	LOCAL CONST Robtarget Tr_meulage_bavure_P179 :=[[-62.25637890625,114.8428984375,23],[0.0433975001230337,-0.0506645555826487,0.757781496955649,-0.649089333345064],[0,0,0,0],[8.999999E+09,8.999999E+09,8.999999E+09,8.999999E+09,8.999999E+09,8.999999E+09]];
	LOCAL CONST Robtarget Tr_meulage_bavure_P180 :=[[-59.10421875,115.2802421875,23],[0.0426624400154122,-0.0495768426742355,0.75636290662596,-0.650874186277744],[0,0,0,0],[8.999999E+09,8.999999E+09,8.999999E+09,8.999999E+09,8.999999E+09,8.999999E+09]];
	LOCAL CONST Robtarget Tr_meulage_bavure_P181 :=[[-53.5016484375,115.9119296875,23],[0.0425676623921922,-0.0492400718100533,0.754898413474392,-0.652603857466726],[0,0,0,0],[8.999999E+09,8.999999E+09,8.999999E+09,8.999999E+09,8.999999E+09,8.999999E+09]];
	LOCAL CONST Robtarget Tr_meulage_bavure_P182 :=[[-50.74237109375,116.2019375,23],[0.0427141238515756,-0.0491877810931781,0.753441246798892,-0.654280026775121],[0,0,0,0],[8.999999E+09,8.999999E+09,8.999999E+09,8.999999E+09,8.999999E+09,8.999999E+09]];
	LOCAL CONST Robtarget Tr_meulage_bavure_P183 :=[[-48.3789375,116.5492578125,23],[0.0426883692327484,-0.0489442555493909,0.752036641826874,-0.65591390618794],[0,0,0,0],[8.999999E+09,8.999999E+09,8.999999E+09,8.999999E+09,8.999999E+09,8.999999E+09]];
	LOCAL CONST Robtarget Tr_meulage_bavure_P184 :=[[-47.19442578125,116.6454453125,23],[0.0421759717467994,-0.0481526058517087,0.750705274857156,-0.657528785878265],[0,0,0,0],[8.999999E+09,8.999999E+09,8.999999E+09,8.999999E+09,8.999999E+09,8.999999E+09]];
	LOCAL CONST Robtarget Tr_meulage_bavure_P185 :=[[-45.17309375,116.962953125,23],[0.0410472512944407,-0.0466708720582419,0.749446158166969,-0.659141417960717],[0,0,0,0],[8.999999E+09,8.999999E+09,8.999999E+09,8.999999E+09,8.999999E+09,8.999999E+09]];
	LOCAL CONST Robtarget Tr_meulage_bavure_P186 :=[[-40.496671875,117.3889140625,23],[0.0393564807118614,-0.0445696628756806,0.748258713502021,-0.66073709616263],[0,0,0,0],[8.999999E+09,8.999999E+09,8.999999E+09,8.999999E+09,8.999999E+09,8.999999E+09]];
	LOCAL CONST Robtarget Tr_meulage_bavure_P187 :=[[-36.24917578125,117.7658671875,23],[0.0372373453158816,-0.0420057842825497,0.74712328336298,-0.662310873878388],[0,0,0,0],[8.999999E+09,8.999999E+09,8.999999E+09,8.999999E+09,8.999999E+09,8.999999E+09]];
	LOCAL CONST Robtarget Tr_meulage_bavure_P188 :=[[-33.85342578125,117.8759453125,23],[0.0348119380921517,-0.0391185229085727,0.746005748898492,-0.663877468168727],[0,0,0,0],[8.999999E+09,8.999999E+09,8.999999E+09,8.999999E+09,8.999999E+09,8.999999E+09]];
	LOCAL CONST Robtarget Tr_meulage_bavure_P189 :=[[-29.71334765625,118.2059609375,23],[0.0321087947450452,-0.0359419945500591,0.744888264782926,-0.665446219702589],[0,0,0,0],[8.999999E+09,8.999999E+09,8.999999E+09,8.999999E+09,8.999999E+09,8.999999E+09]];
	LOCAL CONST Robtarget Tr_meulage_bavure_P190 :=[[-29.433685546875,118.2139296875,23],[0.0290969884705637,-0.0324440804164671,0.743757294915129,-0.667027610499298],[0,0,0,0],[8.999999E+09,8.999999E+09,8.999999E+09,8.999999E+09,8.999999E+09,8.999999E+09]];
	LOCAL CONST Robtarget Tr_meulage_bavure_P191 :=[[-29.069060546875,118.25509375,23],[0.0257723111842326,-0.0286232458964912,0.742595652374559,-0.66863158379258],[0,0,0,0],[8.999999E+09,8.999999E+09,8.999999E+09,8.999999E+09,8.999999E+09,8.999999E+09]];
	LOCAL CONST Robtarget Tr_meulage_bavure_P192 :=[[-24.61538671875,118.4268828125,23],[0.022228048299037,-0.0245871756397275,0.741390680271805,-0.670254611225456],[0,0,0,0],[8.999999E+09,8.999999E+09,8.999999E+09,8.999999E+09,8.999999E+09,8.999999E+09]];
	LOCAL CONST Robtarget Tr_meulage_bavure_P193 :=[[-13.8860166015625,119.1668125,23],[0.0186723067822035,-0.0205674132179465,0.740108243032445,-0.671913770560167],[0,0,0,0],[8.999999E+09,8.999999E+09,8.999999E+09,8.999999E+09,8.999999E+09,8.999999E+09]];
	LOCAL CONST Robtarget Tr_meulage_bavure_P194 :=[[-13.6813046875,119.17703125,23],[0.0153529661705316,-0.0168378187210032,0.738745685652022,-0.673598980270167],[0,0,0,0],[8.999999E+09,8.999999E+09,8.999999E+09,8.999999E+09,8.999999E+09,8.999999E+09]];
	LOCAL CONST Robtarget Tr_meulage_bavure_P195 :=[[-13.675048828125,119.1786171875,23],[0.0124791194821711,-0.013624776925181,0.737304794424137,-0.675307542642514],[0,0,0,0],[8.999999E+09,8.999999E+09,8.999999E+09,8.999999E+09,8.999999E+09,8.999999E+09]];
	LOCAL CONST Robtarget Tr_meulage_bavure_P196 :=[[-13.455474609375,119.18634375,23],[0.0101386523212208,-0.0110181012021846,0.735781987297045,-0.677052934669231],[0,0,0,0],[8.999999E+09,8.999999E+09,8.999999E+09,8.999999E+09,8.999999E+09,8.999999E+09]];
	LOCAL CONST Robtarget Tr_meulage_bavure_P197 :=[[-7.360015625,119.2925703125,23],[0.00825320769388641,-0.00892657242884723,0.734203911666841,-0.678820165405053],[0,0,0,0],[8.999999E+09,8.999999E+09,8.999999E+09,8.999999E+09,8.999999E+09,8.999999E+09]];
	LOCAL CONST Robtarget Tr_meulage_bavure_P198 :=[[-3.48239135742188,119.27084375,23],[0.00660056822057563,-0.0071047154660544,0.732587672437859,-0.680603598072617],[0,0,0,0],[8.999999E+09,8.999999E+09,8.999999E+09,8.999999E+09,8.999999E+09,8.999999E+09]];
	LOCAL CONST Robtarget Tr_meulage_bavure_P199 :=[[2.32504272460938,119.5303359375,23],[0.00486722052895284,-0.00521355358859062,0.730950145915841,-0.682393591125321],[0,0,0,0],[8.999999E+09,8.999999E+09,8.999999E+09,8.999999E+09,8.999999E+09,8.999999E+09]];
	LOCAL CONST Robtarget Tr_meulage_bavure_P200 :=[[2.79562377929688,119.520046875,23],[0.00277067500677587,-0.00295346388518078,0.729309083386742,-0.684172391507196],[0,0,0,0],[8.999999E+09,8.999999E+09,8.999999E+09,8.999999E+09,8.999999E+09,8.999999E+09]];
	LOCAL CONST Robtarget Tr_meulage_bavure_P201 :=[[4.2943115234375,119.581234375,23],[0.000180047461967693,-0.000191012953140271,0.727685334413851,-0.685911062147248],[0,0,0,0],[8.999999E+09,8.999999E+09,8.999999E+09,8.999999E+09,8.999999E+09,8.999999E+09]];
	LOCAL CONST Robtarget Tr_meulage_bavure_P202 :=[[8.9348447265625,119.5882890625,23],[0.00280565935608528,-0.00296283360482063,-0.726097809810713,0.687579319410272],[0,0,0,0],[8.999999E+09,8.999999E+09,8.999999E+09,8.999999E+09,8.999999E+09,8.999999E+09]];
	LOCAL CONST Robtarget Tr_meulage_bavure_P203 :=[[10.968505859375,119.54825,23],[0.00586167132896946,-0.00616291741925017,-0.72456801707136,0.689150816509269],[0,0,0,0],[8.999999E+09,8.999999E+09,8.999999E+09,8.999999E+09,8.999999E+09,8.999999E+09]];
	LOCAL CONST Robtarget Tr_meulage_bavure_P204 :=[[14.89630078125,119.394015625,23],[0.00856705335007749,-0.00897065455951138,-0.723132549518583,0.690597892250205],[0,0,0,0],[8.999999E+09,8.999999E+09,8.999999E+09,8.999999E+09,8.999999E+09,8.999999E+09]];
	LOCAL CONST Robtarget Tr_meulage_bavure_P205 :=[[20.668853515625,119.233,23],[0.010560473092811,-0.0110170912300753,-0.721824674250107,0.691907681524502],[0,0,0,0],[8.999999E+09,8.999999E+09,8.999999E+09,8.999999E+09,8.999999E+09,8.999999E+09]];
	LOCAL CONST Robtarget Tr_meulage_bavure_P206 :=[[22.33157421875,119.166109375,23],[0.01168138525824,-0.0121462082784559,-0.720661370247823,0.693082393583501],[0,0,0,0],[8.999999E+09,8.999999E+09,8.999999E+09,8.999999E+09,8.999999E+09,8.999999E+09]];
	LOCAL CONST Robtarget Tr_meulage_bavure_P207 :=[[22.813384765625,119.130890625,23],[0.01203871621661,-0.0124821682872791,-0.719668639964959,0.694101083011466],[0,0,0,0],[8.999999E+09,8.999999E+09,8.999999E+09,8.999999E+09,8.999999E+09,8.999999E+09]];
	LOCAL CONST Robtarget Tr_meulage_bavure_P208 :=[[26.03826953125,119.161953125,23],[0.0119549919198335,-0.0123665663152091,-0.718863289232462,0.694938643046747],[0,0,0,0],[8.999999E+09,8.999999E+09,8.999999E+09,8.999999E+09,8.999999E+09,8.999999E+09]];
	LOCAL CONST Robtarget Tr_meulage_bavure_P209 :=[[26.30859375,119.1513359375,23],[0.0118491848281992,-0.0122351941419367,-0.718243382528829,0.695583453150492],[0,0,0,0],[8.999999E+09,8.999999E+09,8.999999E+09,8.999999E+09,8.999999E+09,8.999999E+09]];
	LOCAL CONST Robtarget Tr_meulage_bavure_P210 :=[[26.349548828125,119.1507578125,23],[0.0120841139017724,-0.0124621709698921,-0.717804183323817,0.696028607809158],[0,0,0,0],[8.999999E+09,8.999999E+09,8.999999E+09,8.999999E+09,8.999999E+09,8.999999E+09]];
	LOCAL CONST Robtarget Tr_meulage_bavure_P211 :=[[29.7614140625,118.849765625,23],[0.0128620448490422,-0.0132545196420001,-0.717529606068317,0.696283096108764],[0,0,0,0],[8.999999E+09,8.999999E+09,8.999999E+09,8.999999E+09,8.999999E+09,8.999999E+09]];
	LOCAL CONST Robtarget Tr_meulage_bavure_P212 :=[[31.407958984375,118.792171875,23],[0.0142162826118088,-0.0146468680333589,-0.717426178146246,0.696335440341783],[0,0,0,0],[8.999999E+09,8.999999E+09,8.999999E+09,8.999999E+09,8.999999E+09,8.999999E+09]];
	LOCAL CONST Robtarget Tr_meulage_bavure_P213 :=[[36.61441015625,118.40359375,23],[0.0160592402840881,-0.0165499655073942,-0.717475688003378,0.696201721175179],[0,0,0,0],[8.999999E+09,8.999999E+09,8.999999E+09,8.999999E+09,8.999999E+09,8.999999E+09]];
	LOCAL CONST Robtarget Tr_meulage_bavure_P214 :=[[40.49197265625,118.27490625,23],[0.0182751982895402,-0.0188462300699876,-0.717651717591956,0.695907212907685],[0,0,0,0],[8.999999E+09,8.999999E+09,8.999999E+09,8.999999E+09,8.999999E+09,8.999999E+09]];
	LOCAL CONST Robtarget Tr_meulage_bavure_P215 :=[[42.2666640625,118.1718125,23],[0.0207788349409327,-0.0214512327502548,-0.717954080535065,0.695449511377383],[0,0,0,0],[8.999999E+09,8.999999E+09,8.999999E+09,8.999999E+09,8.999999E+09,8.999999E+09]];
	LOCAL CONST Robtarget Tr_meulage_bavure_P216 :=[[43.52847265625,118.1006796875,23],[0.0235383090251198,-0.0243340345160502,-0.718348859509656,0.694858776165046],[0,0,0,0],[8.999999E+09,8.999999E+09,8.999999E+09,8.999999E+09,8.999999E+09,8.999999E+09]];
	LOCAL CONST Robtarget Tr_meulage_bavure_P217 :=[[48.51355078125,117.7652890625,23],[0.026557353073452,-0.0275003853735814,-0.718806879478681,0.694157839267236],[0,0,0,0],[8.999999E+09,8.999999E+09,8.999999E+09,8.999999E+09,8.999999E+09,8.999999E+09]];
	LOCAL CONST Robtarget Tr_meulage_bavure_P218 :=[[49.67135546875,117.659484375,23],[0.0298609904169792,-0.0309787272133096,-0.719309354242342,0.693356108079409],[0,0,0,0],[8.999999E+09,8.999999E+09,8.999999E+09,8.999999E+09,8.999999E+09,8.999999E+09]];
	LOCAL CONST Robtarget Tr_meulage_bavure_P219 :=[[53.21233984375,117.43221875,23],[0.033491058152756,-0.0348139079325028,-0.719824664467954,0.692472954895621],[0,0,0,0],[8.999999E+09,8.999999E+09,8.999999E+09,8.999999E+09,8.999999E+09,8.999999E+09]];
	LOCAL CONST Robtarget Tr_meulage_bavure_P220 :=[[59.14208984375,116.905640625,23],[0.0374768593880479,-0.0390388540160962,-0.72033429845252,0.691512799129874],[0,0,0,0],[8.999999E+09,8.999999E+09,8.999999E+09,8.999999E+09,8.999999E+09,8.999999E+09]];
	LOCAL CONST Robtarget Tr_meulage_bavure_P221 :=[[62.47668359375,116.5752890625,23],[0.041789752182483,-0.0436234769405067,-0.72080230488773,0.690503183295113],[0,0,0,0],[8.999999E+09,8.999999E+09,8.999999E+09,8.999999E+09,8.999999E+09,8.999999E+09]];
	LOCAL CONST Robtarget Tr_meulage_bavure_P222 :=[[66.5614296875,116.081515625,23],[0.0462902130268838,-0.0484217293610688,-0.721213697482429,0.68946599253867],[0,0,0,0],[8.999999E+09,8.999999E+09,8.999999E+09,8.999999E+09,8.999999E+09,8.999999E+09]];
	LOCAL CONST Robtarget Tr_meulage_bavure_P223 :=[[69.88278125,115.7547578125,23],[0.0507075681926275,-0.0531523554276753,-0.721596192911392,0.688405769888854],[0,0,0,0],[8.999999E+09,8.999999E+09,8.999999E+09,8.999999E+09,8.999999E+09,8.999999E+09]];
	LOCAL CONST Robtarget Tr_meulage_bavure_P224 :=[[73.4898046875,115.331453125,23],[0.0546942542132915,-0.0574448811350791,-0.721951545520593,0.687382419114612],[0,0,0,0],[8.999999E+09,8.999999E+09,8.999999E+09,8.999999E+09,8.999999E+09,8.999999E+09]];
	LOCAL CONST Robtarget Tr_meulage_bavure_P225 :=[[74.716734375,115.0784296875,23],[0.0579339284262648,-0.0609602486750725,-0.722302751683078,0.686444639377151],[0,0,0,0],[8.999999E+09,8.999999E+09,8.999999E+09,8.999999E+09,8.999999E+09,8.999999E+09]];
	LOCAL CONST Robtarget Tr_meulage_bavure_P226 :=[[76.93371875,114.7760625,23],[0.0602605795301779,-0.0635194455699666,-0.722685911360463,0.685608500611149],[0,0,0,0],[8.999999E+09,8.999999E+09,8.999999E+09,8.999999E+09,8.999999E+09,8.999999E+09]];
	LOCAL CONST Robtarget Tr_meulage_bavure_P227 :=[[86.0733984375,113.3214140625,23],[0.0617239078973545,-0.0651672003203326,-0.723096863932401,0.684890006181588],[0,0,0,0],[8.999999E+09,8.999999E+09,8.999999E+09,8.999999E+09,8.999999E+09,8.999999E+09]];
	LOCAL CONST Robtarget Tr_meulage_bavure_P228 :=[[86.8890078125,113.1566171875,23],[0.0625462059366649,-0.0661334613382164,-0.723520645014066,0.684274954716877],[0,0,0,0],[8.999999E+09,8.999999E+09,8.999999E+09,8.999999E+09,8.999999E+09,8.999999E+09]];
	LOCAL CONST Robtarget Tr_meulage_bavure_P229 :=[[87.251953125,113.09378125,23],[0.0630269119827303,-0.0667293599938801,-0.723918396754843,0.683752115697367],[0,0,0,0],[8.999999E+09,8.999999E+09,8.999999E+09,8.999999E+09,8.999999E+09,8.999999E+09]];
	LOCAL CONST Robtarget Tr_meulage_bavure_P230 :=[[87.9626484375,112.99203125,23],[0.0634312428074131,-0.0672344832227139,-0.724266199248416,0.683296768855184],[0,0,0,0],[8.999999E+09,8.999999E+09,8.999999E+09,8.999999E+09,8.999999E+09,8.999999E+09]];
	LOCAL CONST Robtarget Tr_meulage_bavure_P231 :=[[93.3311796875,112.030640625,23],[0.0639320549018943,-0.0678358177259327,-0.724567720204724,0.682870861163957],[0,0,0,0],[8.999999E+09,8.999999E+09,8.999999E+09,8.999999E+09,8.999999E+09,8.999999E+09]];
	LOCAL CONST Robtarget Tr_meulage_bavure_P232 :=[[93.9768984375,111.91028125,23],[0.0645980817696378,-0.0686059043245966,-0.72481299252888,0.682470837168019],[0,0,0,0],[8.999999E+09,8.999999E+09,8.999999E+09,8.999999E+09,8.999999E+09,8.999999E+09]];
	LOCAL CONST Robtarget Tr_meulage_bavure_P233 :=[[94.0133671875,111.9046953125,23],[0.0654287527738808,-0.0695441291625365,-0.725000475096411,0.682097502941814],[0,0,0,0],[8.999999E+09,8.999999E+09,8.999999E+09,8.999999E+09,8.999999E+09,8.999999E+09]];
	LOCAL CONST Robtarget Tr_meulage_bavure_P234 :=[[94.076046875,111.892640625,23],[0.0663865651243882,-0.0706134760611833,-0.725146709250839,0.681739547798293],[0,0,0,0],[8.999999E+09,8.999999E+09,8.999999E+09,8.999999E+09,8.999999E+09,8.999999E+09]];
	LOCAL CONST Robtarget Tr_meulage_bavure_P235 :=[[94.187015625,111.8732578125,23],[0.0673897565957632,-0.071729795496014,-0.725273034587947,0.681390110321286],[0,0,0,0],[8.999999E+09,8.999999E+09,8.999999E+09,8.999999E+09,8.999999E+09,8.999999E+09]];
	LOCAL CONST Robtarget Tr_meulage_bavure_P236 :=[[97.91021875,111.1723046875,23],[0.0683393793094796,-0.0727929924441854,-0.725414413490336,0.681032185867223],[0,0,0,0],[8.999999E+09,8.999999E+09,8.999999E+09,8.999999E+09,8.999999E+09,8.999999E+09]];
	LOCAL CONST Robtarget Tr_meulage_bavure_P237 :=[[104.1578359375,110.0602421875,23],[0.0691640964349682,-0.0737272905217292,-0.725580082123736,0.680671843711763],[0,0,0,0],[8.999999E+09,8.999999E+09,8.999999E+09,8.999999E+09,8.999999E+09,8.999999E+09]];
	LOCAL CONST Robtarget Tr_meulage_bavure_P238 :=[[106.742734375,109.5954296875,23],[0.069867288981249,-0.0745393059843067,-0.725784591291777,0.680293452002308],[0,0,0,0],[8.999999E+09,8.999999E+09,8.999999E+09,8.999999E+09,8.999999E+09,8.999999E+09]];
	LOCAL CONST Robtarget Tr_meulage_bavure_P239 :=[[108.946078125,109.0823984375,23],[0.0705682648379406,-0.0753597520797576,-0.726030399452964,0.679868286386716],[0,0,0,0],[8.999999E+09,8.999999E+09,8.999999E+09,8.999999E+09,8.999999E+09,8.999999E+09]];
	LOCAL CONST Robtarget Tr_meulage_bavure_P240 :=[[111.9587421875,108.3916015625,23],[0.071478227758703,-0.0764190215138883,-0.726312485462933,0.679353493821877],[0,0,0,0],[8.999999E+09,8.999999E+09,8.999999E+09,8.999999E+09,8.999999E+09,8.999999E+09]];
	LOCAL CONST Robtarget Tr_meulage_bavure_P241 :=[[116.98425,107.3316953125,23],[0.0728185948770369,-0.0779573259993162,-0.726612015382984,0.678715762793416],[0,0,0,0],[8.999999E+09,8.999999E+09,8.999999E+09,8.999999E+09,8.999999E+09,8.999999E+09]];
	LOCAL CONST Robtarget Tr_meulage_bavure_P242 :=[[119.37615625,106.9286171875,23],[0.0747024713348201,-0.0800980263854046,-0.726909147227233,0.677943167694026],[0,0,0,0],[8.999999E+09,8.999999E+09,8.999999E+09,8.999999E+09,8.999999E+09,8.999999E+09]];
	LOCAL CONST Robtarget Tr_meulage_bavure_P243 :=[[120.3310546875,106.7306484375,23],[0.0770671825316726,-0.0827776894586762,-0.727205350569293,0.677038316203673],[0,0,0,0],[8.999999E+09,8.999999E+09,8.999999E+09,8.999999E+09,8.999999E+09,8.999999E+09]];
	LOCAL CONST Robtarget Tr_meulage_bavure_P244 :=[[121.463625,106.5190703125,23],[0.0796915949839674,-0.0857659743127845,-0.72753514905863,0.676007436514812],[0,0,0,0],[8.999999E+09,8.999999E+09,8.999999E+09,8.999999E+09,8.999999E+09,8.999999E+09]];
	LOCAL CONST Robtarget Tr_meulage_bavure_P245 :=[[125.5679921875,105.588375,23],[0.0822965494182147,-0.0887591416372919,-0.727906997542607,0.674907768260355],[0,0,0,0],[8.999999E+09,8.999999E+09,8.999999E+09,8.999999E+09,8.999999E+09,8.999999E+09]];
	LOCAL CONST Robtarget Tr_meulage_bavure_P246 :=[[126.3385,105.378109375,23],[0.0846657162038379,-0.0915215230583909,-0.728338542426817,0.673779262765145],[0,0,0,0],[8.999999E+09,8.999999E+09,8.999999E+09,8.999999E+09,8.999999E+09,8.999999E+09]];
	LOCAL CONST Robtarget Tr_meulage_bavure_P247 :=[[127.576296875,105.0690625,23],[0.086725938103112,-0.0939680220383543,-0.728824405057627,0.672654152657018],[0,0,0,0],[8.999999E+09,8.999999E+09,8.999999E+09,8.999999E+09,8.999999E+09,8.999999E+09]];
	LOCAL CONST Robtarget Tr_meulage_bavure_P248 :=[[132.538703125,103.8515625,23],[0.0885433965699905,-0.0961628588818879,-0.729338335730027,0.671549226438439],[0,0,0,0],[8.999999E+09,8.999999E+09,8.999999E+09,8.999999E+09,8.999999E+09,8.999999E+09]];
	LOCAL CONST Robtarget Tr_meulage_bavure_P249 :=[[132.940984375,103.7449609375,23],[0.0902923635278784,-0.0982860794839512,-0.729830909733932,0.6704729516283],[0,0,0,0],[8.999999E+09,8.999999E+09,8.999999E+09,8.999999E+09,8.999999E+09,8.999999E+09]];
	LOCAL CONST Robtarget Tr_meulage_bavure_P250 :=[[133.1513125,103.6954375,23],[0.0921721126835679,-0.100543751054332,-0.730239311328871,0.669436930529911],[0,0,0,0],[8.999999E+09,8.999999E+09,8.999999E+09,8.999999E+09,8.999999E+09,8.999999E+09]];
	LOCAL CONST Robtarget Tr_meulage_bavure_P251 :=[[144.677671875,100.6963203125,23],[0.0943708685423752,-0.10313519752154,-0.730514139864084,0.668435757318075],[0,0,0,0],[8.999999E+09,8.999999E+09,8.999999E+09,8.999999E+09,8.999999E+09,8.999999E+09]];
	LOCAL CONST Robtarget Tr_meulage_bavure_P252 :=[[146.309015625,100.2600078125,23],[0.0970895582724477,-0.106272524992245,-0.730595654278941,0.667465173664484],[0,0,0,0],[8.999999E+09,8.999999E+09,8.999999E+09,8.999999E+09,8.999999E+09,8.999999E+09]];
	LOCAL CONST Robtarget Tr_meulage_bavure_P253 :=[[149.755,99.2144765625,23],[0.100467982930273,-0.110099606792247,-0.730427148639799,0.666528650186957],[0,0,0,0],[8.999999E+09,8.999999E+09,8.999999E+09,8.999999E+09,8.999999E+09,8.999999E+09]];
	LOCAL CONST Robtarget Tr_meulage_bavure_P254 :=[[150.8464375,98.8049921875,23],[0.104491902117537,-0.114594138450995,-0.729987100795058,0.665633877215815],[0,0,0,0],[8.999999E+09,8.999999E+09,8.999999E+09,8.999999E+09,8.999999E+09,8.999999E+09]];
	LOCAL CONST Robtarget Tr_meulage_bavure_P255 :=[[154.511234375,97.780484375,23],[0.108876589342561,-0.119438757132208,-0.729312624208754,0.664818296798144],[0,0,0,0],[8.999999E+09,8.999999E+09,8.999999E+09,8.999999E+09,8.999999E+09,8.999999E+09]];
	LOCAL CONST Robtarget Tr_meulage_bavure_P256 :=[[158.105828125,96.761234375,23],[0.113049945403097,-0.123996672016637,-0.728495841137259,0.664182463347891],[0,0,0,0],[8.999999E+09,8.999999E+09,8.999999E+09,8.999999E+09,8.999999E+09,8.999999E+09]];
	LOCAL CONST Robtarget Tr_meulage_bavure_P257 :=[[160.656734375,96.14184375,23],[0.116306712999753,-0.127487992706324,-0.727677158585302,0.663856545573007],[0,0,0,0],[8.999999E+09,8.999999E+09,8.999999E+09,8.999999E+09,8.999999E+09,8.999999E+09]];
	LOCAL CONST Robtarget Tr_meulage_bavure_P258 :=[[162.19371875,95.6184375,23],[0.118092035668419,-0.129308153648255,-0.726995421405591,0.663936239233163],[0,0,0,0],[8.999999E+09,8.999999E+09,8.999999E+09,8.999999E+09,8.999999E+09,8.999999E+09]];
	LOCAL CONST Robtarget Tr_meulage_bavure_P259 :=[[164.91028125,94.8435703125,23],[0.118274965582588,-0.129329702857753,-0.726520291030682,0.664419391044434],[0,0,0,0],[8.999999E+09,8.999999E+09,8.999999E+09,8.999999E+09,8.999999E+09,8.999999E+09]];
	LOCAL CONST Robtarget Tr_meulage_bavure_P260 :=[[166.98015625,94.192109375,23],[0.117243891722456,-0.127988246342763,-0.72618734716399,0.665225386971066],[0,0,0,0],[8.999999E+09,8.999999E+09,8.999999E+09,8.999999E+09,8.999999E+09,8.999999E+09]];
	LOCAL CONST Robtarget Tr_meulage_bavure_P261 :=[[171.675421875,92.646640625,23],[0.11572754801686,-0.126094558058123,-0.72587320873088,0.666194702699495],[0,0,0,0],[8.999999E+09,8.999999E+09,8.999999E+09,8.999999E+09,8.999999E+09,8.999999E+09]];
	LOCAL CONST Robtarget Tr_meulage_bavure_P262 :=[[174.015625,91.8630703125,23],[0.114500012732813,-0.124509658578739,-0.725467910507281,0.66714571334079],[0,0,0,0],[8.999999E+09,8.999999E+09,8.999999E+09,8.999999E+09,8.999999E+09,8.999999E+09]];
	LOCAL CONST Robtarget Tr_meulage_bavure_P263 :=[[175.446171875,91.398984375,23],[0.114108916104908,-0.123841862597972,-0.724912453930014,0.66794032852553],[0,0,0,0],[8.999999E+09,8.999999E+09,8.999999E+09,8.999999E+09,8.999999E+09,8.999999E+09]];
	LOCAL CONST Robtarget Tr_meulage_bavure_P264 :=[[175.904171875,91.263828125,23],[0.114743474933475,-0.124301976981395,-0.724203918231148,0.668514501187043],[0,0,0,0],[8.999999E+09,8.999999E+09,8.999999E+09,8.999999E+09,8.999999E+09,8.999999E+09]];
	LOCAL CONST Robtarget Tr_meulage_bavure_P265 :=[[178.4013125,90.440796875,23],[0.116268429159858,-0.125744534749873,-0.723383533605336,0.668869365175215],[0,0,0,0],[8.999999E+09,8.999999E+09,8.999999E+09,8.999999E+09,8.999999E+09,8.999999E+09]];
	LOCAL CONST Robtarget Tr_meulage_bavure_P266 :=[[182.345765625,89.1579609375,23],[0.118346334643346,-0.12781465659757,-0.722544484889172,0.66901945113096],[0,0,0,0],[8.999999E+09,8.999999E+09,8.999999E+09,8.999999E+09,8.999999E+09,8.999999E+09]];
	LOCAL CONST Robtarget Tr_meulage_bavure_P267 :=[[182.355890625,89.154265625,23],[0.120626665182778,-0.130141775792656,-0.721770309653462,0.668999212214156],[0,0,0,0],[8.999999E+09,8.999999E+09,8.999999E+09,8.999999E+09,8.999999E+09,8.999999E+09]];
	LOCAL CONST Robtarget Tr_meulage_bavure_P268 :=[[182.35778125,89.1534765625,23],[0.122833887482242,-0.132433180424486,-0.721119443046582,0.668849787073931],[0,0,0,0],[8.999999E+09,8.999999E+09,8.999999E+09,8.999999E+09,8.999999E+09,8.999999E+09]];
	LOCAL CONST Robtarget Tr_meulage_bavure_P269 :=[[182.359734375,89.152859375,23],[0.12484680972463,-0.134562502732776,-0.72062029419892,0.668590007813858],[0,0,0,0],[8.999999E+09,8.999999E+09,8.999999E+09,8.999999E+09,8.999999E+09,8.999999E+09]];
	LOCAL CONST Robtarget Tr_meulage_bavure_P270 :=[[186.651421875,87.4858671875,23],[0.126717697865704,-0.136586969306665,-0.720259494978551,0.668216196119549],[0,0,0,0],[8.999999E+09,8.999999E+09,8.999999E+09,8.999999E+09,8.999999E+09,8.999999E+09]];
	LOCAL CONST Robtarget Tr_meulage_bavure_P271 :=[[188.559515625,86.7445703125,23],[0.128587282341396,-0.1386589473087,-0.720004918206395,0.667706466128568],[0,0,0,0],[8.999999E+09,8.999999E+09,8.999999E+09,8.999999E+09,8.999999E+09,8.999999E+09]];
	LOCAL CONST Robtarget Tr_meulage_bavure_P272 :=[[188.560296875,86.744265625,23],[0.130603038526337,-0.140931425656631,-0.719805871718055,0.667053735939083],[0,0,0,0],[8.999999E+09,8.999999E+09,8.999999E+09,8.999999E+09,8.999999E+09,8.999999E+09]];
	LOCAL CONST Robtarget Tr_meulage_bavure_P273 :=[[188.56103125,86.743984375,23],[0.132827486488657,-0.143459006229576,-0.719612865292756,0.666283495570675],[0,0,0,0],[8.999999E+09,8.999999E+09,8.999999E+09,8.999999E+09,8.999999E+09,8.999999E+09]];
	LOCAL CONST Robtarget Tr_meulage_bavure_P274 :=[[188.5729375,86.73946875,23],[0.135174264285544,-0.146146682168728,-0.719433879134541,0.665420137296251],[0,0,0,0],[8.999999E+09,8.999999E+09,8.999999E+09,8.999999E+09,8.999999E+09,8.999999E+09]];
	LOCAL CONST Robtarget Tr_meulage_bavure_P275 :=[[194.580390625,84.4072265625,23],[0.137438881641544,-0.148759849884502,-0.71928091078291,0.664541971781143],[0,0,0,0],[8.999999E+09,8.999999E+09,8.999999E+09,8.999999E+09,8.999999E+09,8.999999E+09]];
	LOCAL CONST Robtarget Tr_meulage_bavure_P276 :=[[195.539921875,84.0454375,23],[0.139384514264984,-0.151026956859485,-0.719177310157503,0.663737005175617],[0,0,0,0],[8.999999E+09,8.999999E+09,8.999999E+09,8.999999E+09,8.999999E+09,8.999999E+09]];
	LOCAL CONST Robtarget Tr_meulage_bavure_P277 :=[[195.803953125,83.922421875,23],[0.140843896039311,-0.152754067464029,-0.719142411616981,0.663071175391734],[0,0,0,0],[8.999999E+09,8.999999E+09,8.999999E+09,8.999999E+09,8.999999E+09,8.999999E+09]];
	LOCAL CONST Robtarget Tr_meulage_bavure_P278 :=[[196.424015625,83.6767265625,23],[0.14180298983553,-0.153905603426694,-0.719146803038966,0.662595542534362],[0,0,0,0],[8.999999E+09,8.999999E+09,8.999999E+09,8.999999E+09,8.999999E+09,8.999999E+09]];
	LOCAL CONST Robtarget Tr_meulage_bavure_P279 :=[[201.51678125,81.5485546875,23],[0.142402663496877,-0.154622811887266,-0.719141166393645,0.662306009538686],[0,0,0,0],[8.999999E+09,8.999999E+09,8.999999E+09,8.999999E+09,8.999999E+09,8.999999E+09]];
	LOCAL CONST Robtarget Tr_meulage_bavure_P280 :=[[204.3700625,80.4995390625,23],[0.142878674299112,-0.155152102512511,-0.719054830498024,0.662173436687046],[0,0,0,0],[8.999999E+09,8.999999E+09,8.999999E+09,8.999999E+09,8.999999E+09,8.999999E+09]];
	LOCAL CONST Robtarget Tr_meulage_bavure_P281 :=[[205.632078125,79.949984375,23],[0.143470255192593,-0.155744309967672,-0.718815492864105,0.662166355990849],[0,0,0,0],[8.999999E+09,8.999999E+09,8.999999E+09,8.999999E+09,8.999999E+09,8.999999E+09]];
	LOCAL CONST Robtarget Tr_meulage_bavure_P282 :=[[209.973015625,77.973171875,23],[0.144354205505574,-0.156581251244078,-0.718363053408254,0.662267845066981],[0,0,0,0],[8.999999E+09,8.999999E+09,8.999999E+09,8.999999E+09,8.999999E+09,8.999999E+09]];
	LOCAL CONST Robtarget Tr_meulage_bavure_P283 :=[[212.1695,76.964875,23],[0.145645067593732,-0.157779480580826,-0.71765821376186,0.662464971159531],[0,0,0,0],[8.999999E+09,8.999999E+09,8.999999E+09,8.999999E+09,8.999999E+09,8.999999E+09]];
	LOCAL CONST Robtarget Tr_meulage_bavure_P284 :=[[214.673578125,75.841921875,23],[0.147371789185419,-0.159371544692817,-0.716701326997084,0.662737862487977],[0,0,0,0],[8.999999E+09,8.999999E+09,8.999999E+09,8.999999E+09,8.999999E+09,8.999999E+09]];
	LOCAL CONST Robtarget Tr_meulage_bavure_P285 :=[[215.543828125,75.423953125,23],[0.149534959261313,-0.161354927903146,-0.715492487825331,0.663079469645687],[0,0,0,0],[8.999999E+09,8.999999E+09,8.999999E+09,8.999999E+09,8.999999E+09,8.999999E+09]];
	LOCAL CONST Robtarget Tr_meulage_bavure_P286 :=[[225.461859375,70.84228125,23],[0.15228784553405,-0.163889501075831,-0.713991876561906,0.663448749899584],[0,0,0,0],[8.999999E+09,8.999999E+09,8.999999E+09,8.999999E+09,8.999999E+09,8.999999E+09]];
	LOCAL CONST Robtarget Tr_meulage_bavure_P287 :=[[226.29015625,70.439453125,23],[0.156016566096224,-0.167386982581166,-0.712107290155373,0.663734612984351],[0,0,0,0],[8.999999E+09,8.999999E+09,8.999999E+09,8.999999E+09,8.999999E+09,8.999999E+09]];
	LOCAL CONST Robtarget Tr_meulage_bavure_P288 :=[[226.441890625,70.3727421875,23],[0.161657150318605,-0.172842246703203,-0.709596030829116,0.663676123223535],[0,0,0,0],[8.999999E+09,8.999999E+09,8.999999E+09,8.999999E+09,8.999999E+09,8.999999E+09]];
	LOCAL CONST Robtarget Tr_meulage_bavure_P289 :=[[226.554875,70.3203125,23],[0.170921299408176,-0.182062360974602,-0.705963474606839,0.662762988289187],[0,0,0,0],[8.999999E+09,8.999999E+09,8.999999E+09,8.999999E+09,8.999999E+09,8.999999E+09]];
	LOCAL CONST Robtarget Tr_meulage_bavure_P290 :=[[230.188421875,68.452484375,23],[0.186264407094151,-0.19761328412548,-0.70034774001563,0.660126960244774],[0,0,0,0],[8.999999E+09,8.999999E+09,8.999999E+09,8.999999E+09,8.999999E+09,8.999999E+09]];
	LOCAL CONST Robtarget Tr_meulage_bavure_P291 :=[[231.19128125,68.0270703125,23],[0.210468767257875,-0.222360769615941,-0.691382664334988,0.65440705803178],[0,0,0,0],[8.999999E+09,8.999999E+09,8.999999E+09,8.999999E+09,8.999999E+09,8.999999E+09]];
	LOCAL CONST Robtarget Tr_meulage_bavure_P292 :=[[234.0234375,66.961484375,23],[0.245666695372288,-0.258440629670158,-0.677149830135849,0.643680373529862],[0,0,0,0],[8.999999E+09,8.999999E+09,8.999999E+09,8.999999E+09,8.999999E+09,8.999999E+09]];
	LOCAL CONST Robtarget Tr_meulage_bavure_P293 :=[[235.546078125,66.28271875,23],[0.291950236957823,-0.305804445250917,-0.655475612127038,0.625779851314929],[0,0,0,0],[8.999999E+09,8.999999E+09,8.999999E+09,8.999999E+09,8.999999E+09,8.999999E+09]];
	LOCAL CONST Robtarget Tr_meulage_bavure_P294 :=[[237.71715625,64.80471875,23],[0.345980377439618,-0.360849099939649,-0.625151518677113,0.599392262375136],[0,0,0,0],[8.999999E+09,8.999999E+09,8.999999E+09,8.999999E+09,8.999999E+09,8.999999E+09]];
	LOCAL CONST Robtarget Tr_meulage_bavure_P295 :=[[238.628484375,64.0985703125,23],[0.401512404121443,-0.417033679688133,-0.587399438452989,0.565537442657432],[0,0,0,0],[8.999999E+09,8.999999E+09,8.999999E+09,8.999999E+09,8.999999E+09,8.999999E+09]];
	LOCAL CONST Robtarget Tr_meulage_bavure_P296 :=[[238.83471875,63.1988203125,23],[0.452322901267873,-0.467944424539678,-0.545892031230331,0.527668360592206],[0,0,0,0],[8.999999E+09,8.999999E+09,8.999999E+09,8.999999E+09,8.999999E+09,8.999999E+09]];
	LOCAL CONST Robtarget Tr_meulage_bavure_P297 :=[[239.54065625,60.9287421875,23],[0.494852816721812,-0.510029297228029,-0.504944966404968,0.489919775732576],[0,0,0,0],[8.999999E+09,8.999999E+09,8.999999E+09,8.999999E+09,8.999999E+09,8.999999E+09]];
	LOCAL CONST Robtarget Tr_meulage_bavure_P298 :=[[238.90209375,58.71240234375,23],[0.528280061960826,-0.542611789662793,-0.467924173813415,0.455565131912705],[0,0,0,0],[8.999999E+09,8.999999E+09,8.999999E+09,8.999999E+09,8.999999E+09,8.999999E+09]];
	LOCAL CONST Robtarget Tr_meulage_bavure_P299 :=[[238.590265625,57.47219921875,23],[0.553335373662547,-0.566588505431125,-0.436817772244424,0.426600121446854],[0,0,0,0],[8.999999E+09,8.999999E+09,8.999999E+09,8.999999E+09,8.999999E+09,8.999999E+09]];
	LOCAL CONST Robtarget Tr_meulage_bavure_P300 :=[[237.893671875,56.071625,23],[0.571297074446085,-0.583388472143138,-0.412466163424204,0.40391732734553],[0,0,0,0],[8.999999E+09,8.999999E+09,8.999999E+09,8.999999E+09,8.999999E+09,8.999999E+09]];
	LOCAL CONST Robtarget Tr_meulage_bavure_P301 :=[[236.861640625,54.1201171875,23],[0.583579557370845,-0.594541794667238,-0.394745607275888,0.387467237517057],[0,0,0,0],[8.999999E+09,8.999999E+09,8.999999E+09,8.999999E+09,8.999999E+09,8.999999E+09]];
	LOCAL CONST Robtarget Tr_meulage_bavure_P302 :=[[235.147578125,50.99142578125,23],[0.591528112684828,-0.601485888975852,-0.382832708544188,0.376494800143609],[0,0,0,0],[8.999999E+09,8.999999E+09,8.999999E+09,8.999999E+09,8.999999E+09,8.999999E+09]];
	LOCAL CONST Robtarget Tr_meulage_bavure_P303 :=[[234.468015625,49.71408203125,23],[0.59636646814935,-0.605499671868604,-0.375458245397209,0.369794928301258],[0,0,0,0],[8.999999E+09,8.999999E+09,8.999999E+09,8.999999E+09,8.999999E+09,8.999999E+09]];
	LOCAL CONST Robtarget Tr_meulage_bavure_P304 :=[[234.070375,49.00653125,23],[0.599118545576107,-0.607641019360047,-0.371260446643969,0.366053330398147],[0,0,0,0],[8.999999E+09,8.999999E+09,8.999999E+09,8.999999E+09,8.999999E+09,8.999999E+09]];
	LOCAL CONST Robtarget Tr_meulage_bavure_P305 :=[[232.982,46.85134765625,23],[0.600566294365692,-0.608692528389672,-0.369070609254375,0.364143402163287],[0,0,0,0],[8.999999E+09,8.999999E+09,8.999999E+09,8.999999E+09,8.999999E+09,8.999999E+09]];
	LOCAL CONST Robtarget Tr_meulage_bavure_P306 :=[[230.236328125,41.5531328125,23],[0.601246025936263,-0.609191571628496,-0.368034698049866,0.363234506048087],[0,0,0,0],[8.999999E+09,8.999999E+09,8.999999E+09,8.999999E+09,8.999999E+09,8.999999E+09]];
	LOCAL CONST Robtarget Tr_meulage_bavure_P307 :=[[228.138796875,37.67785546875,23],[0.60149894341776,-0.609471307200547,-0.367597458866817,0.362788995149016],[0,0,0,0],[8.999999E+09,8.999999E+09,8.999999E+09,8.999999E+09,8.999999E+09,8.999999E+09]];
	LOCAL CONST Robtarget Tr_meulage_bavure_P308 :=[[227.647515625,36.6991875,23],[0.601538517795648,-0.609725951700318,-0.367414433046191,0.362480771656515],[0,0,0,0],[8.999999E+09,8.999999E+09,8.999999E+09,8.999999E+09,8.999999E+09,8.999999E+09]];
	LOCAL CONST Robtarget Tr_meulage_bavure_P309 :=[[227.033015625,35.61612109375,23],[0.601463941385168,-0.610029809508591,-0.367333335467876,0.362175343415832],[0,0,0,0],[8.999999E+09,8.999999E+09,8.999999E+09,8.999999E+09,8.999999E+09,8.999999E+09]];
	LOCAL CONST Robtarget Tr_meulage_bavure_P310 :=[[226.453546875,34.55807421875,23],[0.601323875559455,-0.61040882184473,-0.367284811285392,0.361818371970441],[0,0,0,0],[8.999999E+09,8.999999E+09,8.999999E+09,8.999999E+09,8.999999E+09,8.999999E+09]];
	LOCAL CONST Robtarget Tr_meulage_bavure_P311 :=[[222.681828125,27.470427734375,23],[0.601138129566144,-0.610855076905052,-0.367250443076717,0.361408544809051],[0,0,0,0],[8.999999E+09,8.999999E+09,8.999999E+09,8.999999E+09,8.999999E+09,8.999999E+09]];
	LOCAL CONST Robtarget Tr_meulage_bavure_P312 :=[[219.7761875,21.9488828125,23],[0.60089767770655,-0.611344423057786,-0.367253402836676,0.360977721511867],[0,0,0,0],[8.999999E+09,8.999999E+09,8.999999E+09,8.999999E+09,8.999999E+09,8.999999E+09]];
	LOCAL CONST Robtarget Tr_meulage_bavure_P313 :=[[218.745609375,19.888427734375,23],[0.600593732374037,-0.611840511475639,-0.367323546154104,0.360571448663127],[0,0,0,0],[8.999999E+09,8.999999E+09,8.999999E+09,8.999999E+09,8.999999E+09,8.999999E+09]];
	LOCAL CONST Robtarget Tr_meulage_bavure_P314 :=[[218.2366875,18.98812890625,23],[0.600219263187343,-0.612318662369688,-0.367482565617044,0.360221120674723],[0,0,0,0],[8.999999E+09,8.999999E+09,8.999999E+09,8.999999E+09,8.999999E+09,8.999999E+09]];
	LOCAL CONST Robtarget Tr_meulage_bavure_P315 :=[[215.327328125,13.5820615234375,23],[0.599787051532667,-0.612766172142733,-0.367723199600825,0.359934382306865],[0,0,0,0],[8.999999E+09,8.999999E+09,8.999999E+09,8.999999E+09,8.999999E+09,8.999999E+09]];
	LOCAL CONST Robtarget Tr_meulage_bavure_P316 :=[[212.65240625,8.6597900390625,23],[0.599326303758197,-0.61319369086397,-0.368006567095289,0.359684091506562],[0,0,0,0],[8.999999E+09,8.999999E+09,8.999999E+09,8.999999E+09,8.999999E+09,8.999999E+09]];
	LOCAL CONST Robtarget Tr_meulage_bavure_P317 :=[[211.23540625,5.9966123046875,23],[0.598879090330631,-0.613629377068977,-0.368269313872546,0.359416937862615],[0,0,0,0],[8.999999E+09,8.999999E+09,8.999999E+09,8.999999E+09,8.999999E+09,8.999999E+09]];
	LOCAL CONST Robtarget Tr_meulage_bavure_P318 :=[[209.234015625,2.14840698242188,23],[0.598482704522626,-0.614093592706917,-0.368457697917807,0.359091125800548],[0,0,0,0],[8.999999E+09,8.999999E+09,8.999999E+09,8.999999E+09,8.999999E+09,8.999999E+09]];
	LOCAL CONST Robtarget Tr_meulage_bavure_P319 :=[[206.54271875,-3.07986450195313,23],[0.598155635559902,-0.614574276957813,-0.368557400421948,0.358711215804479],[0,0,0,0],[8.999999E+09,8.999999E+09,8.999999E+09,8.999999E+09,8.999999E+09,8.999999E+09]];
	LOCAL CONST Robtarget Tr_meulage_bavure_P320 :=[[204.57971875,-6.86383056640625,23],[0.597867025447572,-0.615037728341553,-0.368622347157265,0.358331100764647],[0,0,0,0],[8.999999E+09,8.999999E+09,8.999999E+09,8.999999E+09,8.999999E+09,8.999999E+09]];
	LOCAL CONST Robtarget Tr_meulage_bavure_P321 :=[[204.069703125,-7.8434140625,23],[0.59756652899696,-0.615413407596379,-0.368749785890754,0.35805610814321],[0,0,0,0],[8.999999E+09,8.999999E+09,8.999999E+09,8.999999E+09,8.999999E+09,8.999999E+09]];
	LOCAL CONST Robtarget Tr_meulage_bavure_P322 :=[[201.362859375,-12.7850341796875,23],[0.5972042117597,-0.615628186177856,-0.369038341768578,0.35799408953855],[0,0,0,0],[8.999999E+09,8.999999E+09,8.999999E+09,8.999999E+09,8.999999E+09,8.999999E+09]];
	LOCAL CONST Robtarget Tr_meulage_bavure_P323 :=[[197.7320625,-19.72250390625,23],[0.596744410485494,-0.615639798692309,-0.369552658178168,0.358210245043135],[0,0,0,0],[8.999999E+09,8.999999E+09,8.999999E+09,8.999999E+09,8.999999E+09,8.999999E+09]];
	LOCAL CONST Robtarget Tr_meulage_bavure_P324 :=[[196.06928125,-22.846955078125,23],[0.596198525998614,-0.615444856618333,-0.370281117697623,0.358701602917687],[0,0,0,0],[8.999999E+09,8.999999E+09,8.999999E+09,8.999999E+09,8.999999E+09,8.999999E+09]];
	LOCAL CONST Robtarget Tr_meulage_bavure_P325 :=[[193.7264375,-27.16146875,23],[0.595628885421589,-0.615080638126344,-0.371130799141042,0.359393891687736],[0,0,0,0],[8.999999E+09,8.999999E+09,8.999999E+09,8.999999E+09,8.999999E+09,8.999999E+09]];
	LOCAL CONST Robtarget Tr_meulage_bavure_P326 :=[[190.96471875,-32.36828515625,23],[0.595105128360039,-0.614633140154919,-0.371973442934353,0.360155170689591],[0,0,0,0],[8.999999E+09,8.999999E+09,8.999999E+09,8.999999E+09,8.999999E+09,8.999999E+09]];
	LOCAL CONST Robtarget Tr_meulage_bavure_P327 :=[[189.668328125,-34.78494140625,23],[0.594716129997688,-0.614185046446975,-0.372662302133935,0.360849361936163],[0,0,0,0],[8.999999E+09,8.999999E+09,8.999999E+09,8.999999E+09,8.999999E+09,8.999999E+09]];
	LOCAL CONST Robtarget Tr_meulage_bavure_P328 :=[[188.552484375,-37.00442578125,23],[0.594529673614845,-0.613794674386154,-0.373089283396598,0.361379235016672],[0,0,0,0],[8.999999E+09,8.999999E+09,8.999999E+09,8.999999E+09,8.999999E+09,8.999999E+09]];
	LOCAL CONST Robtarget Tr_meulage_bavure_P329 :=[[187.314453125,-39.3024609375,23],[0.594576309018603,-0.613480433801729,-0.373210800102779,0.361710476462738],[0,0,0,0],[8.999999E+09,8.999999E+09,8.999999E+09,8.999999E+09,8.999999E+09,8.999999E+09]];
	LOCAL CONST Robtarget Tr_meulage_bavure_P330 :=[[185.694578125,-42.49502734375,23],[0.594840509861185,-0.613229441364113,-0.373052101102155,0.361865375430714],[0,0,0,0],[8.999999E+09,8.999999E+09,8.999999E+09,8.999999E+09,8.999999E+09,8.999999E+09]];
	LOCAL CONST Robtarget Tr_meulage_bavure_P331 :=[[183.378421875,-46.95462109375,23],[0.595273325691727,-0.61299744880742,-0.372692864489794,0.361916874757033],[0,0,0,0],[8.999999E+09,8.999999E+09,8.999999E+09,8.999999E+09,8.999999E+09,8.999999E+09]];
	LOCAL CONST Robtarget Tr_meulage_bavure_P332 :=[[181.6873125,-50.2353828125,23],[0.59581641235855,-0.61271830826261,-0.37223512036855,0.361966977289646],[0,0,0,0],[8.999999E+09,8.999999E+09,8.999999E+09,8.999999E+09,8.999999E+09,8.999999E+09]];
	LOCAL CONST Robtarget Tr_meulage_bavure_P333 :=[[180.496703125,-52.53855859375,23],[0.596404700565704,-0.612315431419721,-0.37179405551446,0.36213316041551],[0,0,0,0],[8.999999E+09,8.999999E+09,8.999999E+09,8.999999E+09,8.999999E+09,8.999999E+09]];
	LOCAL CONST Robtarget Tr_meulage_bavure_P334 :=[[179.4039375,-54.66871484375,23],[0.596966023347852,-0.6117304207372,-0.371482450346762,0.36251654913577],[0,0,0,0],[8.999999E+09,8.999999E+09,8.999999E+09,8.999999E+09,8.999999E+09,8.999999E+09]];
	LOCAL CONST Robtarget Tr_meulage_bavure_P335 :=[[177.514828125,-58.18369921875,23],[0.597470790505363,-0.610922492471663,-0.371354573992322,0.3631778394397],[0,0,0,0],[8.999999E+09,8.999999E+09,8.999999E+09,8.999999E+09,8.999999E+09,8.999999E+09]];
	LOCAL CONST Robtarget Tr_meulage_bavure_P336 :=[[172.897765625,-66.62578125,23],[0.597938426917615,-0.609915196507573,-0.371373429459774,0.36408085170152],[0,0,0,0],[8.999999E+09,8.999999E+09,8.999999E+09,8.999999E+09,8.999999E+09,8.999999E+09]];
	LOCAL CONST Robtarget Tr_meulage_bavure_P337 :=[[171.1954375,-69.9391015625,23],[0.5984766878218,-0.608822745614949,-0.371354039097867,0.365043416871778],[0,0,0,0],[8.999999E+09,8.999999E+09,8.999999E+09,8.999999E+09,8.999999E+09,8.999999E+09]];
	LOCAL CONST Robtarget Tr_meulage_bavure_P338 :=[[167.682,-76.877640625,23],[0.599271523023736,-0.607831162762065,-0.370987847277633,0.365763497960686],[0,0,0,0],[8.999999E+09,8.999999E+09,8.999999E+09,8.999999E+09,8.999999E+09,8.999999E+09]];
	LOCAL CONST Robtarget Tr_meulage_bavure_P339 :=[[165.8203125,-80.48746875,23],[0.600530131363897,-0.607144358300292,-0.369935660798695,0.365905583966165],[0,0,0,0],[8.999999E+09,8.999999E+09,8.999999E+09,8.999999E+09,8.999999E+09,8.999999E+09]];
	LOCAL CONST Robtarget Tr_meulage_bavure_P340 :=[[165.367,-81.4398828125,23],[0.602379641716574,-0.606891166436327,-0.367986197174384,0.365250650972865],[0,0,0,0],[8.999999E+09,8.999999E+09,8.999999E+09,8.999999E+09,8.999999E+09,8.999999E+09]];
	LOCAL CONST Robtarget Tr_meulage_bavure_P341 :=[[164.5443125,-82.9392578125,23],[0.604782795054275,-0.607036891031052,-0.365193508139137,0.363837443574357],[0,0,0,0],[8.999999E+09,8.999999E+09,8.999999E+09,8.999999E+09,8.999999E+09,8.999999E+09]];
	LOCAL CONST Robtarget Tr_meulage_bavure_P342 :=[[162.21325,-87.17590625,23],[0.607535145214572,-0.607369033032185,-0.361892427507579,0.361991403151138],[0,0,0,0],[8.999999E+09,8.999999E+09,8.999999E+09,8.999999E+09,8.999999E+09,8.999999E+09]];
	LOCAL CONST Robtarget Tr_meulage_bavure_P343 :=[[158.563234375,-93.964984375,23],[0.610323730608498,-0.607577346807641,-0.358601122781731,0.360222079059564],[0,0,0,0],[8.999999E+09,8.999999E+09,8.999999E+09,8.999999E+09,8.999999E+09,8.999999E+09]];
	LOCAL CONST Robtarget Tr_meulage_bavure_P344 :=[[157.13275,-96.60821875,23],[0.612839408371446,-0.607382025815075,-0.355829610279608,0.359026771581137],[0,0,0,0],[8.999999E+09,8.999999E+09,8.999999E+09,8.999999E+09,8.999999E+09,8.999999E+09]];
	LOCAL CONST Robtarget Tr_meulage_bavure_P345 :=[[156.3021875,-98.18434375,23],[0.614901862802277,-0.606625963754836,-0.353878809414897,0.358706603602305],[0,0,0,0],[8.999999E+09,8.999999E+09,8.999999E+09,8.999999E+09,8.999999E+09,8.999999E+09]];
	LOCAL CONST Robtarget Tr_meulage_bavure_P346 :=[[149.948671875,-109.9741328125,23],[0.616486476205011,-0.605320478220127,-0.35277324197074,0.359280646644291],[0,0,0,0],[8.999999E+09,8.999999E+09,8.999999E+09,8.999999E+09,8.999999E+09,8.999999E+09]];
	LOCAL CONST Robtarget Tr_meulage_bavure_P347 :=[[149.3020625,-111.222125,23],[0.617690755263467,-0.603598477114354,-0.352323091152328,0.360548816012686],[0,0,0,0],[8.999999E+09,8.999999E+09,8.999999E+09,8.999999E+09,8.999999E+09,8.999999E+09]];
	LOCAL CONST Robtarget Tr_meulage_bavure_P348 :=[[148.874453125,-111.9904765625,23],[0.618665733996451,-0.601647925107596,-0.352245720185102,0.362209105909328],[0,0,0,0],[8.999999E+09,8.999999E+09,8.999999E+09,8.999999E+09,8.999999E+09,8.999999E+09]];
	LOCAL CONST Robtarget Tr_meulage_bavure_P349 :=[[147.679265625,-114.1219609375,23],[0.619536283467585,-0.599661828340103,-0.352290747339809,0.363966639182405],[0,0,0,0],[8.999999E+09,8.999999E+09,8.999999E+09,8.999999E+09,8.999999E+09,8.999999E+09]];
	LOCAL CONST Robtarget Tr_meulage_bavure_P350 :=[[145.83978125,-117.101515625,23],[0.620401548489368,-0.597781745718546,-0.35227107765951,0.365600862912396],[0,0,0,0],[8.999999E+09,8.999999E+09,8.999999E+09,8.999999E+09,8.999999E+09,8.999999E+09]];
	LOCAL CONST Robtarget Tr_meulage_bavure_P351 :=[[143.49475,-121.2462578125,23],[0.621321427103974,-0.596099369446092,-0.352075011110165,0.366971950589184],[0,0,0,0],[8.999999E+09,8.999999E+09,8.999999E+09,8.999999E+09,8.999999E+09,8.999999E+09]];
	LOCAL CONST Robtarget Tr_meulage_bavure_P352 :=[[141.8126875,-124.3500546875,23],[0.622292228946671,-0.594679982174248,-0.35167896441459,0.368008161026492],[0,0,0,0],[8.999999E+09,8.999999E+09,8.999999E+09,8.999999E+09,8.999999E+09,8.999999E+09]];
	LOCAL CONST Robtarget Tr_meulage_bavure_P353 :=[[140.565796875,-126.8127890625,23],[0.62325513468536,-0.593532657842383,-0.351150322892514,0.368734961585383],[0,0,0,0],[8.999999E+09,8.999999E+09,8.999999E+09,8.999999E+09,8.999999E+09,8.999999E+09]];
	LOCAL CONST Robtarget Tr_meulage_bavure_P354 :=[[139.294859375,-129.0313125,23],[0.624095366593252,-0.592593784826532,-0.350654699588928,0.369295086939968],[0,0,0,0],[8.999999E+09,8.999999E+09,8.999999E+09,8.999999E+09,8.999999E+09,8.999999E+09]];
	LOCAL CONST Robtarget Tr_meulage_bavure_P355 :=[[137.978828125,-131.938109375,23],[0.624654009177447,-0.591758367263694,-0.350426357168808,0.369906436539497],[0,0,0,0],[8.999999E+09,8.999999E+09,8.999999E+09,8.999999E+09,8.999999E+09,8.999999E+09]];
	LOCAL CONST Robtarget Tr_meulage_bavure_P356 :=[[137.96875,-131.957453125,23],[0.624782682949572,-0.590930475217238,-0.350681040799897,0.370770252541066],[0,0,0,0],[8.999999E+09,8.999999E+09,8.999999E+09,8.999999E+09,8.999999E+09,8.999999E+09]];
	LOCAL CONST Robtarget Tr_meulage_bavure_P357 :=[[137.949703125,-131.995703125,23],[0.624412317217918,-0.590077606119387,-0.351511174746379,0.371964475308306],[0,0,0,0],[8.999999E+09,8.999999E+09,8.999999E+09,8.999999E+09,8.999999E+09,8.999999E+09]];
	LOCAL CONST Robtarget Tr_meulage_bavure_P358 :=[[135.40784375,-136.427890625,23],[0.623581938880325,-0.58925624262607,-0.352842420164336,0.373396401376654],[0,0,0,0],[8.999999E+09,8.999999E+09,8.999999E+09,8.999999E+09,8.999999E+09,8.999999E+09]];
	LOCAL CONST Robtarget Tr_meulage_bavure_P359 :=[[134.466609375,-138.346140625,23],[0.62242856660037,-0.588598206416493,-0.3544554474991,0.374828182800211],[0,0,0,0],[8.999999E+09,8.999999E+09,8.999999E+09,8.999999E+09,8.999999E+09,8.999999E+09]];
	LOCAL CONST Robtarget Tr_meulage_bavure_P360 :=[[134.0466875,-139.2799375,23],[0.621121416704301,-0.588264322812558,-0.356085256862142,0.375974150790378],[0,0,0,0],[8.999999E+09,8.999999E+09,8.999999E+09,8.999999E+09,8.999999E+09,8.999999E+09]];
	LOCAL CONST Robtarget Tr_meulage_bavure_P361 :=[[133.17303125,-140.80175,23],[0.619809170320105,-0.588371223582879,-0.357513643367062,0.376616370399772],[0,0,0,0],[8.999999E+09,8.999999E+09,8.999999E+09,8.999999E+09,8.999999E+09,8.999999E+09]];
	LOCAL CONST Robtarget Tr_meulage_bavure_P362 :=[[131.86615625,-143.383296875,23],[0.618565640936541,-0.588946424218623,-0.358647085909467,0.376684118355833],[0,0,0,0],[8.999999E+09,8.999999E+09,8.999999E+09,8.999999E+09,8.999999E+09,8.999999E+09]];
	LOCAL CONST Robtarget Tr_meulage_bavure_P363 :=[[131.544671875,-143.900140625,23],[0.617364929904112,-0.589946735548578,-0.359533634901461,0.37624321643667],[0,0,0,0],[8.999999E+09,8.999999E+09,8.999999E+09,8.999999E+09,8.999999E+09,8.999999E+09]];
	LOCAL CONST Robtarget Tr_meulage_bavure_P364 :=[[131.0465078125,-144.800515625,23],[0.616144126663892,-0.591263070585177,-0.360291153336647,0.37545263531786],[0,0,0,0],[8.999999E+09,8.999999E+09,8.999999E+09,8.999999E+09,8.999999E+09,8.999999E+09]];
	LOCAL CONST Robtarget Tr_meulage_bavure_P365 :=[[128.491640625,-149.462078125,23],[0.614843489236258,-0.592762781250768,-0.361045294724983,0.374494411259485],[0,0,0,0],[8.999999E+09,8.999999E+09,8.999999E+09,8.999999E+09,8.999999E+09,8.999999E+09]];
	LOCAL CONST Robtarget Tr_meulage_bavure_P366 :=[[126.1275,-154.528984375,23],[0.613427714221348,-0.594365248031995,-0.361871510638103,0.373477443958178],[0,0,0,0],[8.999999E+09,8.999999E+09,8.999999E+09,8.999999E+09,8.999999E+09,8.999999E+09]];
	LOCAL CONST Robtarget Tr_meulage_bavure_P367 :=[[125.9691796875,-154.83228125,23],[0.611914102773742,-0.596025643924273,-0.362770386427466,0.372440880332073],[0,0,0,0],[8.999999E+09,8.999999E+09,8.999999E+09,8.999999E+09,8.999999E+09,8.999999E+09]];
	LOCAL CONST Robtarget Tr_meulage_bavure_P368 :=[[123.9113125,-158.798859375,23],[0.610358466348196,-0.597722216229869,-0.363688772344218,0.371377397875917],[0,0,0,0],[8.999999E+09,8.999999E+09,8.999999E+09,8.999999E+09,8.999999E+09,8.999999E+09]];
	LOCAL CONST Robtarget Tr_meulage_bavure_P369 :=[[122.6449609375,-161.21334375,23],[0.608804605776085,-0.5994451021539,-0.364581543822902,0.370273978822757],[0,0,0,0],[8.999999E+09,8.999999E+09,8.999999E+09,8.999999E+09,8.999999E+09,8.999999E+09]];
	LOCAL CONST Robtarget Tr_meulage_bavure_P370 :=[[122.51165625,-161.48296875,23],[0.607281762019995,-0.601161249530756,-0.365431922509032,0.369152439504147],[0,0,0,0],[8.999999E+09,8.999999E+09,8.999999E+09,8.999999E+09,8.999999E+09,8.999999E+09]];
	LOCAL CONST Robtarget Tr_meulage_bavure_P371 :=[[121.02484375,-164.35209375,23],[0.605792366795316,-0.602832281817099,-0.366256903892271,0.368055333724382],[0,0,0,0],[8.999999E+09,8.999999E+09,8.999999E+09,8.999999E+09,8.999999E+09,8.999999E+09]];
	LOCAL CONST Robtarget Tr_meulage_bavure_P372 :=[[116.380859375,-173.294921875,23],[0.604339649989507,-0.604426902860253,-0.367069887747645,0.367016898872864],[0,0,0,0],[8.999999E+09,8.999999E+09,8.999999E+09,8.999999E+09,8.999999E+09,8.999999E+09]];
	LOCAL CONST Robtarget Tr_meulage_bavure_P373 :=[[115.6409296875,-174.713890625,23],[0.602944163587668,-0.60592289711816,-0.367860704856743,0.366052291572943],[0,0,0,0],[8.999999E+09,8.999999E+09,8.999999E+09,8.999999E+09,8.999999E+09,8.999999E+09]];
	LOCAL CONST Robtarget Tr_meulage_bavure_P374 :=[[114.1279921875,-177.56259375,23],[0.601625812863237,-0.607319958495692,-0.368608698577571,0.365152675797932],[0,0,0,0],[8.999999E+09,8.999999E+09,8.999999E+09,8.999999E+09,8.999999E+09,8.999999E+09]];
	LOCAL CONST Robtarget Tr_meulage_bavure_P375 :=[[109.4513515625,-186.506609375,23],[0.600385411844571,-0.60861572454795,-0.369315739388538,0.364321481273197],[0,0,0,0],[8.999999E+09,8.999999E+09,8.999999E+09,8.999999E+09,8.999999E+09,8.999999E+09]];
	LOCAL CONST Robtarget Tr_meulage_bavure_P376 :=[[108.4268828125,-188.458703125,23],[0.599177711767558,-0.609761821726402,-0.370060428876233,0.363637002333139],[0,0,0,0],[8.999999E+09,8.999999E+09,8.999999E+09,8.999999E+09,8.999999E+09,8.999999E+09]];
	LOCAL CONST Robtarget Tr_meulage_bavure_P377 :=[[108.223453125,-188.801953125,23],[0.597924418780761,-0.610680344443884,-0.37097519956498,0.36322624856047],[0,0,0,0],[8.999999E+09,8.999999E+09,8.999999E+09,8.999999E+09,8.999999E+09,8.999999E+09]];
	LOCAL CONST Robtarget Tr_meulage_bavure_P378 :=[[105.705625,-193.336890625,23],[0.596517430529864,-0.611266139223228,-0.372240876523167,0.363259400371749],[0,0,0,0],[8.999999E+09,8.999999E+09,8.999999E+09,8.999999E+09,8.999999E+09,8.999999E+09]];
	LOCAL CONST Robtarget Tr_meulage_bavure_P379 :=[[101.5655859375,-200.7506875,23],[0.59485996243784,-0.61143312314165,-0.374013181837981,0.363875391892786],[0,0,0,0],[8.999999E+09,8.999999E+09,8.999999E+09,8.999999E+09,8.999999E+09,8.999999E+09]];
	LOCAL CONST Robtarget Tr_meulage_bavure_P380 :=[[98.17984375,-207.054015625,23],[0.592972487689151,-0.611222458173416,-0.376243213100121,0.365009287641128],[0,0,0,0],[8.999999E+09,8.999999E+09,8.999999E+09,8.999999E+09,8.999999E+09,8.999999E+09]];
	LOCAL CONST Robtarget Tr_meulage_bavure_P381 :=[[97.604859375,-208.15246875,23],[0.591056407097362,-0.610858997578545,-0.378579812330341,0.366307158546508],[0,0,0,0],[8.999999E+09,8.999999E+09,8.999999E+09,8.999999E+09,8.999999E+09,8.999999E+09]];
	LOCAL CONST Robtarget Tr_meulage_bavure_P382 :=[[96.052859375,-211.20721875,23],[0.589602090012172,-0.610877277042716,-0.380191571384328,0.366950537394988],[0,0,0,0],[8.999999E+09,8.999999E+09,8.999999E+09,8.999999E+09,8.999999E+09,8.999999E+09]];
	LOCAL CONST Robtarget Tr_meulage_bavure_P383 :=[[93.876796875,-215.554640625,23],[0.589435944812638,-0.612139838035832,-0.379701427379883,0.365618533034061],[0,0,0,0],[8.999999E+09,8.999999E+09,8.999999E+09,8.999999E+09,8.999999E+09,8.999999E+09]];
	LOCAL CONST Robtarget Tr_meulage_bavure_P384 :=[[92.8142734375,-217.610765625,23],[0.591526357925115,-0.615682363947228,-0.375415794742584,0.360686533796309],[0,0,0,0],[8.999999E+09,8.999999E+09,8.999999E+09,8.999999E+09,8.999999E+09,8.999999E+09]];
	LOCAL CONST Robtarget Tr_meulage_bavure_P385 :=[[92.00375,-219.249296875,23],[0.596661472355205,-0.622361448180502,-0.36570384199059,0.350602360486789],[0,0,0,0],[8.999999E+09,8.999999E+09,8.999999E+09,8.999999E+09,8.999999E+09,8.999999E+09]];
	LOCAL CONST Robtarget Tr_meulage_bavure_P386 :=[[91.4444609375,-220.7653125,23],[0.605064538950082,-0.632443649514328,-0.349469016147819,0.334340157095732],[0,0,0,0],[8.999999E+09,8.999999E+09,8.999999E+09,8.999999E+09,8.999999E+09,8.999999E+09]];
	LOCAL CONST Robtarget Tr_meulage_bavure_P387 :=[[91.329375,-221.03240625,23],[0.616182861646669,-0.645358755029341,-0.326537729356398,0.311775351217298],[0,0,0,0],[8.999999E+09,8.999999E+09,8.999999E+09,8.999999E+09,8.999999E+09,8.999999E+09]];
	LOCAL CONST Robtarget Tr_meulage_bavure_P388 :=[[88.64075,-226.41875,23],[0.628924013659979,-0.659968180176956,-0.2975129673466,0.283518289456537],[0,0,0,0],[8.999999E+09,8.999999E+09,8.999999E+09,8.999999E+09,8.999999E+09,8.999999E+09]];
	LOCAL CONST Robtarget Tr_meulage_bavure_P389 :=[[88.2015703125,-227.09140625,23],[0.642233778731465,-0.675176562260016,-0.262919561462365,0.250091358170348],[0,0,0,0],[8.999999E+09,8.999999E+09,8.999999E+09,8.999999E+09,8.999999E+09,8.999999E+09]];
	LOCAL CONST Robtarget Tr_meulage_bavure_P390 :=[[87.6403828125,-227.443453125,23],[0.655489947681885,-0.690329793523963,-0.222069566701044,0.210862069150364],[0,0,0,0],[8.999999E+09,8.999999E+09,8.999999E+09,8.999999E+09,8.999999E+09,8.999999E+09]];
	LOCAL CONST Robtarget Tr_meulage_bavure_P391 :=[[86.9151640625,-227.967796875,23],[0.668232353026627,-0.704903849997751,-0.172620705117455,0.163640388631897],[0,0,0,0],[8.999999E+09,8.999999E+09,8.999999E+09,8.999999E+09,8.999999E+09,8.999999E+09]];
	LOCAL CONST Robtarget Tr_meulage_bavure_P392 :=[[86.285890625,-228.445171875,23],[0.679199699031414,-0.717562844873643,-0.112020626333748,0.106031654557852],[0,0,0,0],[8.999999E+09,8.999999E+09,8.999999E+09,8.999999E+09,8.999999E+09,8.999999E+09]];
	LOCAL CONST Robtarget Tr_meulage_bavure_P393 :=[[85.749296875,-228.884625,23],[0.685836169933842,-0.725583173327494,-0.0408382158490568,0.0386011233094115],[0,0,0,0],[8.999999E+09,8.999999E+09,8.999999E+09,8.999999E+09,8.999999E+09,8.999999E+09]];
	LOCAL CONST Robtarget Tr_meulage_bavure_P394 :=[[82.9827578125,-228.534,23],[0.68572841206225,-0.726355775880424,0.0339808088621371,-0.0320801553114656],[0,0,0,0],[8.999999E+09,8.999999E+09,8.999999E+09,8.999999E+09,8.999999E+09,8.999999E+09]];
	LOCAL CONST Robtarget Tr_meulage_bavure_P395 :=[[82.6018984375,-228.50490625,23],[0.679353955958623,-0.720356978559851,0.101757695761688,-0.0959656048632183],[0,0,0,0],[8.999999E+09,8.999999E+09,8.999999E+09,8.999999E+09,8.999999E+09,8.999999E+09]];
	LOCAL CONST Robtarget Tr_meulage_bavure_P396 :=[[82.2412109375,-228.248875,23],[0.669967975904944,-0.711023129411504,0.155398258225526,-0.14642541461159],[0,0,0,0],[8.999999E+09,8.999999E+09,8.999999E+09,8.999999E+09,8.999999E+09,8.999999E+09]];
	LOCAL CONST Robtarget Tr_meulage_bavure_P397 :=[[80.2981875,-227.036390625,23],[0.660704391289296,-0.701664599316537,0.194177924774438,-0.182842639795253],[0,0,0,0],[8.999999E+09,8.999999E+09,8.999999E+09,8.999999E+09,8.999999E+09,8.999999E+09]];
	LOCAL CONST Robtarget Tr_meulage_bavure_P398 :=[[79.5094921875,-226.343609375,23],[0.653050539974788,-0.693874170092481,0.220951552400353,-0.207952013236185],[0,0,0,0],[8.999999E+09,8.999999E+09,8.999999E+09,8.999999E+09,8.999999E+09,8.999999E+09]];
	LOCAL CONST Robtarget Tr_meulage_bavure_P399 :=[[78.45065625,-225.310421875,23],[0.6472341485305,-0.687897065524321,0.239218568406757,-0.22507789928922],[0,0,0,0],[8.999999E+09,8.999999E+09,8.999999E+09,8.999999E+09,8.999999E+09,8.999999E+09]];
	LOCAL CONST Robtarget Tr_meulage_bavure_P400 :=[[77.5211171875,-224.47896875,23],[0.642968320483474,-0.683439247130644,0.251781848471526,-0.236872191521971],[0,0,0,0],[8.999999E+09,8.999999E+09,8.999999E+09,8.999999E+09,8.999999E+09,8.999999E+09]];
	LOCAL CONST Robtarget Tr_meulage_bavure_P401 :=[[76.9691484375,-223.91896875,23],[0.639879313640029,-0.680113377310592,0.26057248901841,-0.245157573706171],[0,0,0,0],[8.999999E+09,8.999999E+09,8.999999E+09,8.999999E+09,8.999999E+09,8.999999E+09]];
	LOCAL CONST Robtarget Tr_meulage_bavure_P402 :=[[74.2886640625,-220.9869375,23],[0.637672741756993,-0.677616986573435,0.266789049121338,-0.251062337271422],[0,0,0,0],[8.999999E+09,8.999999E+09,8.999999E+09,8.999999E+09,8.999999E+09,8.999999E+09]];
	LOCAL CONST Robtarget Tr_meulage_bavure_P403 :=[[72.9103359375,-219.65515625,23],[0.63613514420905,-0.675739192710477,0.271178832676306,-0.255285452866865],[0,0,0,0],[8.999999E+09,8.999999E+09,8.999999E+09,8.999999E+09,8.999999E+09,8.999999E+09]];
	LOCAL CONST Robtarget Tr_meulage_bavure_P404 :=[[68.806640625,-215.527734375,23],[0.635086398832137,-0.674304713324809,0.274295232124961,-0.258341915375512],[0,0,0,0],[8.999999E+09,8.999999E+09,8.999999E+09,8.999999E+09,8.999999E+09,8.999999E+09]];
	LOCAL CONST Robtarget Tr_meulage_bavure_P405 :=[[62.0220625,-208.755734375,23],[0.634410716998139,-0.673197736457045,0.276480189990059,-0.260550483265873],[0,0,0,0],[8.999999E+09,8.999999E+09,8.999999E+09,8.999999E+09,8.999999E+09,8.999999E+09]];
	LOCAL CONST Robtarget Tr_meulage_bavure_P406 :=[[58.56121875,-205.267859375,23],[0.63400648199346,-0.672325408686159,0.27800458928837,-0.262159825220934],[0,0,0,0],[8.999999E+09,8.999999E+09,8.999999E+09,8.999999E+09,8.999999E+09,8.999999E+09]];
	LOCAL CONST Robtarget Tr_meulage_bavure_P407 :=[[56.6865546875,-203.365125,23],[0.633792831293324,-0.671617834008434,0.279071202867967,-0.263354126173935],[0,0,0,0],[8.999999E+09,8.999999E+09,8.999999E+09,8.999999E+09,8.999999E+09,8.999999E+09]];
	LOCAL CONST Robtarget Tr_meulage_bavure_P408 :=[[55.1875625,-201.806125,23],[0.633710888346319,-0.671028815485629,0.279819169259009,-0.264257585121922],[0,0,0,0],[8.999999E+09,8.999999E+09,8.999999E+09,8.999999E+09,8.999999E+09,8.999999E+09]];
	LOCAL CONST Robtarget Tr_meulage_bavure_P409 :=[[53.33056640625,-199.943578125,23],[0.633709194555404,-0.67051571285868,0.280369775462135,-0.264979479493922],[0,0,0,0],[8.999999E+09,8.999999E+09,8.999999E+09,8.999999E+09,8.999999E+09,8.999999E+09]];
	LOCAL CONST Robtarget Tr_meulage_bavure_P410 :=[[51.210265625,-197.795046875,23],[0.633757591104653,-0.670054045734295,0.280793061561639,-0.265582657737987],[0,0,0,0],[8.999999E+09,8.999999E+09,8.999999E+09,8.999999E+09,8.999999E+09,8.999999E+09]];
	LOCAL CONST Robtarget Tr_meulage_bavure_P411 :=[[47.50116015625,-194.06184375,23],[0.633842314977253,-0.669638676150633,0.281114701575651,-0.266087368556903],[0,0,0,0],[8.999999E+09,8.999999E+09,8.999999E+09,8.999999E+09,8.999999E+09,8.999999E+09]];
	LOCAL CONST Robtarget Tr_meulage_bavure_P412 :=[[43.991484375,-190.50859375,23],[0.633963442126396,-0.669286625707838,0.281317320097953,-0.266470133614958],[0,0,0,0],[8.999999E+09,8.999999E+09,8.999999E+09,8.999999E+09,8.999999E+09,8.999999E+09]];
	LOCAL CONST Robtarget Tr_meulage_bavure_P413 :=[[38.1468203125,-184.54321875,23],[0.634133200567133,-0.669016597089722,0.281364797687685,-0.266694070761128],[0,0,0,0],[8.999999E+09,8.999999E+09,8.999999E+09,8.999999E+09,8.999999E+09,8.999999E+09]];
	LOCAL CONST Robtarget Tr_meulage_bavure_P414 :=[[35.9768984375,-182.271609375,23],[0.634351700996416,-0.668831389218795,0.281254543232091,-0.266755270144599],[0,0,0,0],[8.999999E+09,8.999999E+09,8.999999E+09,8.999999E+09,8.999999E+09,8.999999E+09]];
	LOCAL CONST Robtarget Tr_meulage_bavure_P415 :=[[31.27362109375,-177.2996875,23],[0.634591803205445,-0.668712574756256,0.281044057775507,-0.266703905588947],[0,0,0,0],[8.999999E+09,8.999999E+09,8.999999E+09,8.999999E+09,8.999999E+09,8.999999E+09]];
	LOCAL CONST Robtarget Tr_meulage_bavure_P416 :=[[23.23678515625,-169.187015625,23],[0.634811497663405,-0.668619163205618,0.280835228025953,-0.266635240971959],[0,0,0,0],[8.999999E+09,8.999999E+09,8.999999E+09,8.999999E+09,8.999999E+09,8.999999E+09]];
	LOCAL CONST Robtarget Tr_meulage_bavure_P417 :=[[22.062775390625,-168.017296875,23],[0.634968530903519,-0.668512414983091,0.280727983916072,-0.266641922476793],[0,0,0,0],[8.999999E+09,8.999999E+09,8.999999E+09,8.999999E+09,8.999999E+09,8.999999E+09]];
	LOCAL CONST Robtarget Tr_meulage_bavure_P418 :=[[21.56253125,-167.508578125,23],[0.63504456791037,-0.668376199842311,0.280764972825024,-0.266763345095322],[0,0,0,0],[8.999999E+09,8.999999E+09,8.999999E+09,8.999999E+09,8.999999E+09,8.999999E+09]];
	LOCAL CONST Robtarget Tr_meulage_bavure_P419 :=[[8.383880859375,-153.8000625,23],[0.635052132698886,-0.668225887967205,0.280912389840672,-0.266966628324664],[0,0,0,0],[8.999999E+09,8.999999E+09,8.999999E+09,8.999999E+09,8.999999E+09,8.999999E+09]];
	LOCAL CONST Robtarget Tr_meulage_bavure_P420 :=[[8.0638427734375,-153.467046875,23],[0.635024212294037,-0.668096959159077,0.281086741949393,-0.267172128903837],[0,0,0,0],[8.999999E+09,8.999999E+09,8.999999E+09,8.999999E+09,8.999999E+09,8.999999E+09]];
	LOCAL CONST Robtarget Tr_meulage_bavure_P421 :=[[6.970458984375,-152.33534375,23],[0.634993766868028,-0.668024807792717,0.281204922668016,-0.267300511932789],[0,0,0,0],[8.999999E+09,8.999999E+09,8.999999E+09,8.999999E+09,8.999999E+09,8.999999E+09]];
	LOCAL CONST Robtarget Tr_meulage_bavure_P422 :=[[4.91180419921875,-150.261953125,23],[0.634976225692153,-0.668024221364001,0.281230032232622,-0.267317229985661],[0,0,0,0],[8.999999E+09,8.999999E+09,8.999999E+09,8.999999E+09,8.999999E+09,8.999999E+09]];
	LOCAL CONST Robtarget Tr_meulage_bavure_P423 :=[[0.50537109375,-145.87303125,23],[0.634968618694908,-0.668087772967172,0.281174030902968,-0.26723537421199],[0,0,0,0],[8.999999E+09,8.999999E+09,8.999999E+09,8.999999E+09,8.999999E+09,8.999999E+09]];
	LOCAL CONST Robtarget Tr_meulage_bavure_P424 :=[[-2.5142822265625,-142.788,23],[0.634958382056523,-0.668199820024187,0.281070775485691,-0.267088136658443],[0,0,0,0],[8.999999E+09,8.999999E+09,8.999999E+09,8.999999E+09,8.999999E+09,8.999999E+09]];
	LOCAL CONST Robtarget Tr_meulage_bavure_P425 :=[[-4.16226171875,-141.127328125,23],[0.634937548351542,-0.668348771118902,0.280943440717684,-0.266898881516756],[0,0,0,0],[8.999999E+09,8.999999E+09,8.999999E+09,8.999999E+09,8.999999E+09,8.999999E+09]];
	LOCAL CONST Robtarget Tr_meulage_bavure_P426 :=[[-6.9866640625,-138.21509375,23],[0.634912553913432,-0.668532647902049,0.280784979448425,-0.266664476239984],[0,0,0,0],[8.999999E+09,8.999999E+09,8.999999E+09,8.999999E+09,8.999999E+09,8.999999E+09]];
	LOCAL CONST Robtarget Tr_meulage_bavure_P427 :=[[-15.706482421875,-129.192046875,23],[0.634895405451963,-0.66875803837555,0.280571474422639,-0.266364708594027],[0,0,0,0],[8.999999E+09,8.999999E+09,8.999999E+09,8.999999E+09,8.999999E+09,8.999999E+09]];
	LOCAL CONST Robtarget Tr_meulage_bavure_P428 :=[[-17.284119140625,-127.578703125,23],[0.634892670068794,-0.669027537917633,0.280290693343183,-0.265989808500223],[0,0,0,0],[8.999999E+09,8.999999E+09,8.999999E+09,8.999999E+09,8.999999E+09,8.999999E+09]];
	LOCAL CONST Robtarget Tr_meulage_bavure_P429 :=[[-20.572205078125,-124.222015625,23],[0.634901097558417,-0.669330610393216,0.27995796204366,-0.265557281576165],[0,0,0,0],[8.999999E+09,8.999999E+09,8.999999E+09,8.999999E+09,8.999999E+09,8.999999E+09]];
	LOCAL CONST Robtarget Tr_meulage_bavure_P430 :=[[-24.6383046875,-120.106015625,23],[0.63490541012216,-0.669645570468371,0.279617441882863,-0.265111328208709],[0,0,0,0],[8.999999E+09,8.999999E+09,8.999999E+09,8.999999E+09,8.999999E+09,8.999999E+09]];
	LOCAL CONST Robtarget Tr_meulage_bavure_P431 :=[[-27.08834765625,-117.671203125,23],[0.634890135827596,-0.669950188256773,0.279314498481349,-0.264697320767784],[0,0,0,0],[8.999999E+09,8.999999E+09,8.999999E+09,8.999999E+09,8.999999E+09,8.999999E+09]];
	LOCAL CONST Robtarget Tr_meulage_bavure_P432 :=[[-30.53274609375,-114.320828125,23],[0.634849159940023,-0.670236423374151,0.279066506071341,-0.264332302405905],[0,0,0,0],[8.999999E+09,8.999999E+09,8.999999E+09,8.999999E+09,8.999999E+09,8.999999E+09]];
	LOCAL CONST Robtarget Tr_meulage_bavure_P433 :=[[-32.92599609375,-111.968640625,23],[0.634797092098068,-0.670515607476437,0.278840991842225,-0.263987070256833],[0,0,0,0],[8.999999E+09,8.999999E+09,8.999999E+09,8.999999E+09,8.999999E+09,8.999999E+09]];
	LOCAL CONST Robtarget Tr_meulage_bavure_P434 :=[[-34.352140625,-110.570359375,23],[0.6347655546915,-0.670821436343292,0.278557283406435,-0.263585149393402],[0,0,0,0],[8.999999E+09,8.999999E+09,8.999999E+09,8.999999E+09,8.999999E+09,8.999999E+09]];
	LOCAL CONST Robtarget Tr_meulage_bavure_P435 :=[[-38.74209765625,-106.158828125,23],[0.634791127072671,-0.671196033766624,0.278118023265371,-0.263033219158196],[0,0,0,0],[8.999999E+09,8.999999E+09,8.999999E+09,8.999999E+09,8.999999E+09,8.999999E+09]];
	LOCAL CONST Robtarget Tr_meulage_bavure_P436 :=[[-40.5563046875,-104.313125,23],[0.63490935429755,-0.6716757611095,0.277432371446258,-0.26224618784102],[0,0,0,0],[8.999999E+09,8.999999E+09,8.999999E+09,8.999999E+09,8.999999E+09,8.999999E+09]];
	LOCAL CONST Robtarget Tr_meulage_bavure_P437 :=[[-42.07171484375,-102.7633671875,23],[0.635140973337646,-0.672287888441827,0.276438539494954,-0.261164072804883],[0,0,0,0],[8.999999E+09,8.999999E+09,8.999999E+09,8.999999E+09,8.999999E+09,8.999999E+09]];
	LOCAL CONST Robtarget Tr_meulage_bavure_P438 :=[[-47.26516796875,-97.63134375,23],[0.635497574885513,-0.673053222969112,0.275092569331458,-0.259742698962143],[0,0,0,0],[8.999999E+09,8.999999E+09,8.999999E+09,8.999999E+09,8.999999E+09,8.999999E+09]];
	LOCAL CONST Robtarget Tr_meulage_bavure_P439 :=[[-52.4834296875,-92.5108359375,23],[0.635992541534395,-0.67398906838904,0.273349123138836,-0.25793890688286],[0,0,0,0],[8.999999E+09,8.999999E+09,8.999999E+09,8.999999E+09,8.999999E+09,8.999999E+09]];
	LOCAL CONST Robtarget Tr_meulage_bavure_P440 :=[[-55.64529296875,-89.3565234375,23],[0.63664042733376,-0.675118412339705,0.271151315846734,-0.255697202798129],[0,0,0,0],[8.999999E+09,8.999999E+09,8.999999E+09,8.999999E+09,8.999999E+09,8.999999E+09]];
	LOCAL CONST Robtarget Tr_meulage_bavure_P441 :=[[-57.77978515625,-87.28459375,23],[0.637463288832554,-0.676469942466569,0.268419846310136,-0.252942203748017],[0,0,0,0],[8.999999E+09,8.999999E+09,8.999999E+09,8.999999E+09,8.999999E+09,8.999999E+09]];
	LOCAL CONST Robtarget Tr_meulage_bavure_P442 :=[[-62.9189765625,-82.356265625,23],[0.638475889237702,-0.678066480821458,0.265085497209506,-0.249607823630827],[0,0,0,0],[8.999999E+09,8.999999E+09,8.999999E+09,8.999999E+09,8.999999E+09,8.999999E+09]];
	LOCAL CONST Robtarget Tr_meulage_bavure_P443 :=[[-65.390625,-80.054140625,23],[0.63967855536182,-0.679911223318349,0.26111526659223,-0.24566418495261],[0,0,0,0],[8.999999E+09,8.999999E+09,8.999999E+09,8.999999E+09,8.999999E+09,8.999999E+09]];
	LOCAL CONST Robtarget Tr_meulage_bavure_P444 :=[[-66.9117734375,-78.71171875,23],[0.641050772495705,-0.681986398975452,0.25652603575906,-0.241128288827539],[0,0,0,0],[8.999999E+09,8.999999E+09,8.999999E+09,8.999999E+09,8.999999E+09,8.999999E+09]];
	LOCAL CONST Robtarget Tr_meulage_bavure_P445 :=[[-68.4579140625,-77.3150625,23],[0.642552855934404,-0.684250958581479,0.251390329051981,-0.236070657791274],[0,0,0,0],[8.999999E+09,8.999999E+09,8.999999E+09,8.999999E+09,8.999999E+09,8.999999E+09]];
	LOCAL CONST Robtarget Tr_meulage_bavure_P446 :=[[-70.4374375,-75.583828125,23],[0.644133188906594,-0.686647328076875,0.245824419847128,-0.230604068482614],[0,0,0,0],[8.999999E+09,8.999999E+09,8.999999E+09,8.999999E+09,8.999999E+09,8.999999E+09]];
	LOCAL CONST Robtarget Tr_meulage_bavure_P447 :=[[-72.639375,-73.7899453125,23],[0.645744510276746,-0.689123282192309,0.239940619428412,-0.224836893183157],[0,0,0,0],[8.999999E+09,8.999999E+09,8.999999E+09,8.999999E+09,8.999999E+09,8.999999E+09]];
	LOCAL CONST Robtarget Tr_meulage_bavure_P448 :=[[-75.8875703125,-71.2039375,23],[0.64735587314854,-0.691639022454705,0.233818866850479,-0.218848289056025],[0,0,0,0],[8.999999E+09,8.999999E+09,8.999999E+09,8.999999E+09,8.999999E+09,8.999999E+09]];
	LOCAL CONST Robtarget Tr_meulage_bavure_P449 :=[[-77.985109375,-69.6199765625,23],[0.648964906220088,-0.694182042838219,0.227460438625532,-0.21264428220855],[0,0,0,0],[8.999999E+09,8.999999E+09,8.999999E+09,8.999999E+09,8.999999E+09,8.999999E+09]];
	LOCAL CONST Robtarget Tr_meulage_bavure_P450 :=[[-79.6962578125,-68.31103125,23],[0.650595436194931,-0.696770607209369,0.22077412234055,-0.206143363308584],[0,0,0,0],[8.999999E+09,8.999999E+09,8.999999E+09,8.999999E+09,8.999999E+09,8.999999E+09]];
	LOCAL CONST Robtarget Tr_meulage_bavure_P451 :=[[-82.728,-66.1858359375,23],[0.652288614045467,-0.699435300343164,0.21360433617971,-0.199205954192482],[0,0,0,0],[8.999999E+09,8.999999E+09,8.999999E+09,8.999999E+09,8.999999E+09,8.999999E+09]];
	LOCAL CONST Robtarget Tr_meulage_bavure_P452 :=[[-86.9236484375,-63.3616953125,23],[0.654088411833945,-0.702213343918629,0.205752934423605,-0.191652026086967],[0,0,0,0],[8.999999E+09,8.999999E+09,8.999999E+09,8.999999E+09,8.999999E+09,8.999999E+09]];
	LOCAL CONST Robtarget Tr_meulage_bavure_P453 :=[[-90.6213984375,-61.1728359375,23],[0.656019762036596,-0.705119444199149,0.197058832045428,-0.183337006473388],[0,0,0,0],[8.999999E+09,8.999999E+09,8.999999E+09,8.999999E+09,8.999999E+09,8.999999E+09]];
	LOCAL CONST Robtarget Tr_meulage_bavure_P454 :=[[-93.6788046875,-59.28190625,23],[0.658088702958667,-0.708144086783622,0.18740427260372,-0.174157543624845],[0,0,0,0],[8.999999E+09,8.999999E+09,8.999999E+09,8.999999E+09,8.999999E+09,8.999999E+09]];
	LOCAL CONST Robtarget Tr_meulage_bavure_P455 :=[[-97.18740625,-57.62183984375,23],[0.660278565058086,-0.711258118974761,0.176720873920473,-0.164054373419618],[0,0,0,0],[8.999999E+09,8.999999E+09,8.999999E+09,8.999999E+09,8.999999E+09,8.999999E+09]];
	LOCAL CONST Robtarget Tr_meulage_bavure_P456 :=[[-98.288265625,-57.077421875,23],[0.662549296844525,-0.714406852810528,0.165016712275502,-0.153038434969668],[0,0,0,0],[8.999999E+09,8.999999E+09,8.999999E+09,8.999999E+09,8.999999E+09,8.999999E+09]];
	LOCAL CONST Robtarget Tr_meulage_bavure_P457 :=[[-98.5339375,-56.99624609375,23],[0.664831963758228,-0.717505893054702,0.152430331980226,-0.14124003430172],[0,0,0,0],[8.999999E+09,8.999999E+09,8.999999E+09,8.999999E+09,8.999999E+09,8.999999E+09]];
	LOCAL CONST Robtarget Tr_meulage_bavure_P458 :=[[-104.47409375,-54.51058984375,23],[0.667023564976952,-0.720430991761291,0.139338919167681,-0.129009361987661],[0,0,0,0],[8.999999E+09,8.999999E+09,8.999999E+09,8.999999E+09,8.999999E+09,8.999999E+09]];
	LOCAL CONST Robtarget Tr_meulage_bavure_P459 :=[[-106.81246875,-53.807890625,23],[0.668994574745117,-0.723028244373478,0.126445302725919,-0.116995735898179],[0,0,0,0],[8.999999E+09,8.999999E+09,8.999999E+09,8.999999E+09,8.999999E+09,8.999999E+09]];
	LOCAL CONST Robtarget Tr_meulage_bavure_P460 :=[[-110.1105078125,-52.7649375,23],[0.670617504093768,-0.725155839774868,0.114731694996361,-0.106102824687717],[0,0,0,0],[8.999999E+09,8.999999E+09,8.999999E+09,8.999999E+09,8.999999E+09,8.999999E+09]];
	LOCAL CONST Robtarget Tr_meulage_bavure_P461 :=[[-111.331265625,-52.42426953125,23],[0.671803490174236,-0.726711285746012,0.105317546262951,-0.0973601161063645],[0,0,0,0],[8.999999E+09,8.999999E+09,8.999999E+09,8.999999E+09,8.999999E+09,8.999999E+09]];
	LOCAL CONST Robtarget Tr_meulage_bavure_P462 :=[[-112.5874296875,-52.10264453125,23],[0.672516314317457,-0.727648172014264,0.0992091554007234,-0.0916923564199298],[0,0,0,0],[8.999999E+09,8.999999E+09,8.999999E+09,8.999999E+09,8.999999E+09,8.999999E+09]];
	LOCAL CONST Robtarget Tr_meulage_bavure_P463 :=[[-114.8395078125,-51.604125,23],[0.672753462777654,-0.727960456092208,0.0970871344159712,-0.0897242498859454],[0,0,0,0],[8.999999E+09,8.999999E+09,8.999999E+09,8.999999E+09,8.999999E+09,8.999999E+09]];
	LOCAL CONST Robtarget Tr_meulage_bavure_degg1 :=[[-117.45213604728,-61.2246619458437,23.7870467460616],[0.672753462777654,-0.727960456092208,0.0970871344159712,-0.0897242498859454],[0,0,0,0],[8.999999E+09,8.999999E+09,8.999999E+09,8.999999E+09,8.999999E+09,8.999999E+09]];
	LOCAL CONST Robtarget Tr_meulage_bavure_degg2 :=[[-167.092072508103,-244.014863916874,38.7409349212322],[0.672753462777654,-0.727960456092208,0.0970871344159712,-0.0897242498859454],[0,0,0,0],[8.999999E+09,8.999999E+09,8.999999E+09,8.999999E+09,8.999999E+09,8.999999E+09]];
	LOCAL PROC Tr_pick()
		!!Programme Tr_pick - 22/03/2023 14:34:50;
		 CONST Robtarget Ppick :=[[35.5086084969221,-17.0271592880655,52.6514389635504],[-0.0232270152452578,0.999396228594326,0.00190741360654813,-0.0257690862773143],[0,0,0,0],[8.999999E+09,8.999999E+09,8.999999E+09,8.999999E+09,8.999999E+09,8.999999E+09]];
		 VAR Pose Ref :=[[0,0,0],[1,0,0,0]];
		LocalisationPieceTable 60 \model:=0;
		MoveJ Reltool(Ppick,0,0,-200),V1000,Z0,Tool_Prehenseur \Wobj:=Wobj_vision;
		MoveL Reltool(Ppick,0,0,-100),V500,Z0,Tool_Prehenseur \Wobj:=Wobj_vision;
		MoveL Reltool(Ppick,0,0,-10),V200,Z0,Tool_Prehenseur \Wobj:=Wobj_vision;
		MoveL Ppick,V100,Fine,Tool_Prehenseur \Wobj:=Wobj_vision;
		Gripper_Close;
		MoveL Reltool(Ppick,0,0,-200),V500,Z0,Tool_Prehenseur \Wobj:=Wobj_vision;
		LocalisationPiecePrehenseur 60 \model:=0,Ref;
	ENDPROC
	LOCAL PROC Tr_Cut()
		!!Programme Tr_Cut - 22/03/2023 14:34:50;
		confJ \off;
		confL \off;
		Tool := ToolOffset(Tool_M2_D490_S180);
		MoveAbsJ [[0,-40,40,0,90,0],[8.999999E+09,8.999999E+09,8.999999E+09,8.999999E+09,8.999999E+09,8.999999E+09]] ,V1000,Z0,Tool_M2_D490_S180 \Wobj:=Wobj_Part_0;
		Movej Reltool(Coupe_0,-200,0,-71.932453125),V1000,Z0,Tool_M2_D490_S180 \Wobj:=Wobj_Part_0;
		MoveL Reltool(Coupe_0,0,0,-71.932453125),V500,Z0,Tool_M2_D490_S180 \Wobj:=Wobj_Part_0;
		MoveL Reltool(Coupe_0,0,0,-61.932453125),vitesse_Tronconnage,Z0,Tool_M2_D490_S180 \Wobj:=Wobj_Part_0;
		MoveL Coupe_0,vitesse_Tronconnage,Fine,Tool_M2_D490_S180 \Wobj:=Wobj_Part_0;
		MoveL Reltool(Coupe_0,0,0,61.932453125),vitesse_Tronconnage,Z0,Tool_M2_D490_S180 \Wobj:=Wobj_Part_0;
		MoveL Reltool(Coupe_0,-200,0,61.932453125),V500,Z0,Tool_M2_D490_S180 \Wobj:=Wobj_Part_0;
		MoveAbsJ [[0,-40,40,0,90,0],[8.999999E+09,8.999999E+09,8.999999E+09,8.999999E+09,8.999999E+09,8.999999E+09]] ,V1000,Z0,Tool_M2_D490_S180 \Wobj:=Wobj_Part_0;
		Movej Reltool(Coupe_1,-200,0,-61.67085546875),V1000,Z0,Tool_M2_D490_S180 \Wobj:=Wobj_Part_0;
		MoveL Reltool(Coupe_1,0,0,-61.67085546875),V500,Z0,Tool_M2_D490_S180 \Wobj:=Wobj_Part_0;
		MoveL Reltool(Coupe_1,0,0,-51.67085546875),vitesse_Tronconnage,Z0,Tool_M2_D490_S180 \Wobj:=Wobj_Part_0;
		MoveL Coupe_1,vitesse_Tronconnage,Fine,Tool_M2_D490_S180 \Wobj:=Wobj_Part_0;
		MoveL Reltool(Coupe_1,0,0,51.67085546875),vitesse_Tronconnage,Z0,Tool_M2_D490_S180 \Wobj:=Wobj_Part_0;
		MoveL Reltool(Coupe_1,-200,0,51.67085546875),V500,Z0,Tool_M2_D490_S180 \Wobj:=Wobj_Part_0;
	ENDPROC
	LOCAL PROC Tr_meulage_motif_1()
		!!Programme Tr_meulage_motif_1 - 22/03/2023 14:34:50;
		 CONST Speeddata vitesse_Meulage :=[50, 500, 0, 0];
		confJ \off;
		confL \off;
		Tool := ToolOffset(Tool_M1_D500_S0);
		MoveAbsJ [[0,-40,40,0,90,0],[8.999999E+09,8.999999E+09,8.999999E+09,8.999999E+09,8.999999E+09,8.999999E+09]] ,V1000,Z0,Tool_M1_D500_S0 \Wobj:=Wobj_Part_0;
		MoveJ Tr_meulage_motif_1_App1,V2000,Z100,Tool,\Wobj:=Wobj_Part_0;
		MoveJ Tr_meulage_motif_1_App2,V500,Z0,Tool,\Wobj:=Wobj_Part_0;
		MoveL Tr_meulage_motif_1_P0,[12.5,500,0,0],z0,Tool \wobj:=Wobj_Part_0;
		MoveL Tr_meulage_motif_1_P1,[12.5,500,0,0],z0,Tool \wobj:=Wobj_Part_0;
		MoveL Tr_meulage_motif_1_P2,[12.5,500,0,0],z0,Tool \wobj:=Wobj_Part_0;
		MoveL Tr_meulage_motif_1_P3,[12.5,500,0,0],z0,Tool \wobj:=Wobj_Part_0;
		MoveL Tr_meulage_motif_1_P4,[12.5,500,0,0],z0,Tool \wobj:=Wobj_Part_0;
		MoveL Tr_meulage_motif_1_P5,[12.5,500,0,0],z0,Tool \wobj:=Wobj_Part_0;
		MoveL Tr_meulage_motif_1_P6,[12.5,500,0,0],z0,Tool \wobj:=Wobj_Part_0;
		MoveL Tr_meulage_motif_1_P7,[12.5,500,0,0],z0,Tool \wobj:=Wobj_Part_0;
		MoveL Tr_meulage_motif_1_P8,[12.5,500,0,0],z0,Tool \wobj:=Wobj_Part_0;
		MoveL Tr_meulage_motif_1_P9,[12.5,500,0,0],z0,Tool \wobj:=Wobj_Part_0;
		MoveL Tr_meulage_motif_1_P10,[12.5,500,0,0],z0,Tool \wobj:=Wobj_Part_0;
		MoveL Tr_meulage_motif_1_P11,[12.5,500,0,0],z0,Tool \wobj:=Wobj_Part_0;
		MoveL Tr_meulage_motif_1_P12,[12.5,500,0,0],z0,Tool \wobj:=Wobj_Part_0;
		MoveL Tr_meulage_motif_1_P13,[12.5,500,0,0],z0,Tool \wobj:=Wobj_Part_0;
		MoveL Tr_meulage_motif_1_P14,[12.5,500,0,0],z0,Tool \wobj:=Wobj_Part_0;
		MoveL Tr_meulage_motif_1_P15,[12.5,500,0,0],z0,Tool \wobj:=Wobj_Part_0;
		MoveL Tr_meulage_motif_1_P16,[12.5,500,0,0],z0,Tool \wobj:=Wobj_Part_0;
		MoveL Tr_meulage_motif_1_P17,[12.5,500,0,0],z0,Tool \wobj:=Wobj_Part_0;
		MoveL Tr_meulage_motif_1_P18,[12.5,500,0,0],z0,Tool \wobj:=Wobj_Part_0;
		MoveL Tr_meulage_motif_1_P19,[12.5,500,0,0],z0,Tool \wobj:=Wobj_Part_0;
		MoveL Tr_meulage_motif_1_P20,[12.5,500,0,0],z0,Tool \wobj:=Wobj_Part_0;
		MoveL Tr_meulage_motif_1_P21,[12.5,500,0,0],z0,Tool \wobj:=Wobj_Part_0;
		MoveL Tr_meulage_motif_1_P22,[12.5,500,0,0],z0,Tool \wobj:=Wobj_Part_0;
		MoveL Tr_meulage_motif_1_P23,[12.5,500,0,0],z0,Tool \wobj:=Wobj_Part_0;
		MoveL Tr_meulage_motif_1_P24,[12.5,500,0,0],z0,Tool \wobj:=Wobj_Part_0;
		MoveL Tr_meulage_motif_1_P25,[12.5,500,0,0],z0,Tool \wobj:=Wobj_Part_0;
		MoveL Tr_meulage_motif_1_P26,[12.5,500,0,0],z0,Tool \wobj:=Wobj_Part_0;
		MoveL Tr_meulage_motif_1_P27,[12.5,500,0,0],z0,Tool \wobj:=Wobj_Part_0;
		MoveL Tr_meulage_motif_1_P28,[12.5,500,0,0],z0,Tool \wobj:=Wobj_Part_0;
		MoveL Tr_meulage_motif_1_P29,[12.5,500,0,0],z0,Tool \wobj:=Wobj_Part_0;
		MoveL Tr_meulage_motif_1_P30,[12.5,500,0,0],z0,Tool \wobj:=Wobj_Part_0;
		MoveL Tr_meulage_motif_1_P31,[12.5,500,0,0],z0,Tool \wobj:=Wobj_Part_0;
		MoveL Tr_meulage_motif_1_P32,[12.5,500,0,0],z0,Tool \wobj:=Wobj_Part_0;
		MoveL Tr_meulage_motif_1_P33,[12.5,500,0,0],z0,Tool \wobj:=Wobj_Part_0;
		MoveL Tr_meulage_motif_1_P34,[12.5,500,0,0],z0,Tool \wobj:=Wobj_Part_0;
		MoveL Tr_meulage_motif_1_P35,[12.5,500,0,0],z0,Tool \wobj:=Wobj_Part_0;
		MoveL Tr_meulage_motif_1_P36,[12.5,500,0,0],z0,Tool \wobj:=Wobj_Part_0;
		MoveL Tr_meulage_motif_1_P37,[12.5,500,0,0],z0,Tool \wobj:=Wobj_Part_0;
		MoveL Tr_meulage_motif_1_P38,[12.5,500,0,0],z0,Tool \wobj:=Wobj_Part_0;
		MoveL Tr_meulage_motif_1_P39,[12.5,500,0,0],z0,Tool \wobj:=Wobj_Part_0;
		MoveL Tr_meulage_motif_1_P40,[12.5,500,0,0],z0,Tool \wobj:=Wobj_Part_0;
		MoveL Tr_meulage_motif_1_P41,[12.5,500,0,0],z0,Tool \wobj:=Wobj_Part_0;
		MoveL Tr_meulage_motif_1_P42,[12.5,500,0,0],z0,Tool \wobj:=Wobj_Part_0;
		MoveL Tr_meulage_motif_1_P43,[12.5,500,0,0],z0,Tool \wobj:=Wobj_Part_0;
		MoveL Tr_meulage_motif_1_P44,[12.5,500,0,0],z0,Tool \wobj:=Wobj_Part_0;
		MoveL Tr_meulage_motif_1_P45,[12.5,500,0,0],z0,Tool \wobj:=Wobj_Part_0;
		MoveL Tr_meulage_motif_1_P46,[12.5,500,0,0],z0,Tool \wobj:=Wobj_Part_0;
		MoveL Tr_meulage_motif_1_P47,[12.5,500,0,0],z0,Tool \wobj:=Wobj_Part_0;
		MoveL Tr_meulage_motif_1_P48,[12.5,500,0,0],z0,Tool \wobj:=Wobj_Part_0;
		MoveL Tr_meulage_motif_1_P49,[12.5,500,0,0],z0,Tool \wobj:=Wobj_Part_0;
		MoveL Tr_meulage_motif_1_P50,[12.5,500,0,0],z0,Tool \wobj:=Wobj_Part_0;
		MoveL Tr_meulage_motif_1_P51,[12.5,500,0,0],z0,Tool \wobj:=Wobj_Part_0;
		MoveL Tr_meulage_motif_1_P52,[12.5,500,0,0],z0,Tool \wobj:=Wobj_Part_0;
		MoveL Tr_meulage_motif_1_P53,[12.5,500,0,0],z0,Tool \wobj:=Wobj_Part_0;
		MoveL Tr_meulage_motif_1_P54,[12.5,500,0,0],z0,Tool \wobj:=Wobj_Part_0;
		MoveL Tr_meulage_motif_1_P55,[12.5,500,0,0],z0,Tool \wobj:=Wobj_Part_0;
		MoveL Tr_meulage_motif_1_P56,[12.5,500,0,0],z0,Tool \wobj:=Wobj_Part_0;
		MoveL Tr_meulage_motif_1_P57,[12.5,500,0,0],z0,Tool \wobj:=Wobj_Part_0;
		MoveL Tr_meulage_motif_1_P58,[12.5,500,0,0],z0,Tool \wobj:=Wobj_Part_0;
		MoveL Tr_meulage_motif_1_P59,[12.5,500,0,0],z0,Tool \wobj:=Wobj_Part_0;
		MoveL Tr_meulage_motif_1_P60,[12.5,500,0,0],z0,Tool \wobj:=Wobj_Part_0;
		MoveL Tr_meulage_motif_1_P61,[12.5,500,0,0],z0,Tool \wobj:=Wobj_Part_0;
		MoveL Tr_meulage_motif_1_P62,[12.5,500,0,0],z0,Tool \wobj:=Wobj_Part_0;
		MoveL Tr_meulage_motif_1_P63,[12.5,500,0,0],z0,Tool \wobj:=Wobj_Part_0;
		MoveL Tr_meulage_motif_1_P64,[12.5,500,0,0],z0,Tool \wobj:=Wobj_Part_0;
		MoveL Tr_meulage_motif_1_P65,[12.5,500,0,0],z0,Tool \wobj:=Wobj_Part_0;
		MoveL Tr_meulage_motif_1_P66,[12.5,500,0,0],z0,Tool \wobj:=Wobj_Part_0;
		MoveL Tr_meulage_motif_1_P67,[12.5,500,0,0],z0,Tool \wobj:=Wobj_Part_0;
		MoveL Tr_meulage_motif_1_P68,[12.5,500,0,0],z0,Tool \wobj:=Wobj_Part_0;
		MoveL Tr_meulage_motif_1_P69,[12.5,500,0,0],z0,Tool \wobj:=Wobj_Part_0;
		MoveL Tr_meulage_motif_1_P70,[12.5,500,0,0],z0,Tool \wobj:=Wobj_Part_0;
		MoveL Tr_meulage_motif_1_P71,[12.5,500,0,0],z0,Tool \wobj:=Wobj_Part_0;
		MoveL Tr_meulage_motif_1_P72,[12.5,500,0,0],z0,Tool \wobj:=Wobj_Part_0;
		MoveL Tr_meulage_motif_1_P73,[12.5,500,0,0],z0,Tool \wobj:=Wobj_Part_0;
		MoveL Tr_meulage_motif_1_P74,[12.5,500,0,0],z0,Tool \wobj:=Wobj_Part_0;
		MoveL Tr_meulage_motif_1_P75,[12.5,500,0,0],z0,Tool \wobj:=Wobj_Part_0;
		MoveL Tr_meulage_motif_1_P76,[12.5,500,0,0],z0,Tool \wobj:=Wobj_Part_0;
		MoveL Tr_meulage_motif_1_P77,[12.5,500,0,0],z0,Tool \wobj:=Wobj_Part_0;
		MoveL Tr_meulage_motif_1_P78,[12.5,500,0,0],z0,Tool \wobj:=Wobj_Part_0;
		MoveL Tr_meulage_motif_1_P79,[12.5,500,0,0],z0,Tool \wobj:=Wobj_Part_0;
		MoveL Tr_meulage_motif_1_P80,[12.5,500,0,0],z0,Tool \wobj:=Wobj_Part_0;
		MoveL Tr_meulage_motif_1_P81,[12.5,500,0,0],z0,Tool \wobj:=Wobj_Part_0;
		MoveL Tr_meulage_motif_1_P82,[12.5,500,0,0],z0,Tool \wobj:=Wobj_Part_0;
		MoveL Tr_meulage_motif_1_P83,[12.5,500,0,0],z0,Tool \wobj:=Wobj_Part_0;
		MoveL Tr_meulage_motif_1_P84,[12.5,500,0,0],z0,Tool \wobj:=Wobj_Part_0;
		MoveL Tr_meulage_motif_1_P85,[12.5,500,0,0],z0,Tool \wobj:=Wobj_Part_0;
		MoveL Tr_meulage_motif_1_P86,[12.5,500,0,0],z0,Tool \wobj:=Wobj_Part_0;
		MoveL Tr_meulage_motif_1_P87,[12.5,500,0,0],z0,Tool \wobj:=Wobj_Part_0;
		MoveL Tr_meulage_motif_1_P88,[12.5,500,0,0],z0,Tool \wobj:=Wobj_Part_0;
		MoveL Tr_meulage_motif_1_P89,[12.5,500,0,0],z0,Tool \wobj:=Wobj_Part_0;
		MoveL Tr_meulage_motif_1_P90,[12.5,500,0,0],z0,Tool \wobj:=Wobj_Part_0;
		MoveL Tr_meulage_motif_1_P91,[12.5,500,0,0],z0,Tool \wobj:=Wobj_Part_0;
		MoveL Tr_meulage_motif_1_P92,[12.5,500,0,0],z0,Tool \wobj:=Wobj_Part_0;
		MoveL Tr_meulage_motif_1_P93,[12.5,500,0,0],z0,Tool \wobj:=Wobj_Part_0;
		MoveL Tr_meulage_motif_1_P94,[12.5,500,0,0],z0,Tool \wobj:=Wobj_Part_0;
		MoveL Tr_meulage_motif_1_P95,[12.5,500,0,0],z0,Tool \wobj:=Wobj_Part_0;
		MoveL Tr_meulage_motif_1_P96,[12.5,500,0,0],z0,Tool \wobj:=Wobj_Part_0;
		MoveL Tr_meulage_motif_1_P97,[12.5,500,0,0],z0,Tool \wobj:=Wobj_Part_0;
		MoveL Tr_meulage_motif_1_P98,[12.5,500,0,0],z0,Tool \wobj:=Wobj_Part_0;
		MoveL Tr_meulage_motif_1_P99,[12.5,500,0,0],z0,Tool \wobj:=Wobj_Part_0;
		MoveL Tr_meulage_motif_1_P100,[12.5,500,0,0],z0,Tool \wobj:=Wobj_Part_0;
		MoveL Tr_meulage_motif_1_P101,[12.5,500,0,0],z0,Tool \wobj:=Wobj_Part_0;
		MoveL Tr_meulage_motif_1_P102,[12.5,500,0,0],z0,Tool \wobj:=Wobj_Part_0;
		MoveL Tr_meulage_motif_1_P103,[12.5,500,0,0],z0,Tool \wobj:=Wobj_Part_0;
		MoveL Tr_meulage_motif_1_P104,[12.5,500,0,0],z0,Tool \wobj:=Wobj_Part_0;
		MoveL Tr_meulage_motif_1_P105,[12.5,500,0,0],z0,Tool \wobj:=Wobj_Part_0;
		MoveL Tr_meulage_motif_1_P106,[12.5,500,0,0],z0,Tool \wobj:=Wobj_Part_0;
		MoveL Tr_meulage_motif_1_P107,[12.5,500,0,0],z0,Tool \wobj:=Wobj_Part_0;
		MoveL Tr_meulage_motif_1_P108,[12.5,500,0,0],z0,Tool \wobj:=Wobj_Part_0;
		MoveL Tr_meulage_motif_1_P109,[12.5,500,0,0],z0,Tool \wobj:=Wobj_Part_0;
		MoveL Tr_meulage_motif_1_P110,[12.5,500,0,0],z0,Tool \wobj:=Wobj_Part_0;
		MoveL Tr_meulage_motif_1_P111,[12.5,500,0,0],z0,Tool \wobj:=Wobj_Part_0;
		MoveL Tr_meulage_motif_1_P112,[12.5,500,0,0],z0,Tool \wobj:=Wobj_Part_0;
		MoveL Tr_meulage_motif_1_P113,[12.5,500,0,0],z0,Tool \wobj:=Wobj_Part_0;
		MoveL Tr_meulage_motif_1_P114,[12.5,500,0,0],z0,Tool \wobj:=Wobj_Part_0;
		MoveL Tr_meulage_motif_1_P115,[12.5,500,0,0],z0,Tool \wobj:=Wobj_Part_0;
		MoveL Tr_meulage_motif_1_P116,[12.5,500,0,0],z0,Tool \wobj:=Wobj_Part_0;
		MoveL Tr_meulage_motif_1_P117,[12.5,500,0,0],z0,Tool \wobj:=Wobj_Part_0;
		MoveL Tr_meulage_motif_1_P118,[12.5,500,0,0],z0,Tool \wobj:=Wobj_Part_0;
		MoveL Tr_meulage_motif_1_P119,[12.5,500,0,0],z0,Tool \wobj:=Wobj_Part_0;
		MoveL Tr_meulage_motif_1_P120,[12.5,500,0,0],z0,Tool \wobj:=Wobj_Part_0;
		MoveL Tr_meulage_motif_1_P121,[12.5,500,0,0],z0,Tool \wobj:=Wobj_Part_0;
		MoveL Tr_meulage_motif_1_P122,[12.5,500,0,0],z0,Tool \wobj:=Wobj_Part_0;
		MoveL Tr_meulage_motif_1_P123,[12.5,500,0,0],z0,Tool \wobj:=Wobj_Part_0;
		MoveL Tr_meulage_motif_1_P124,[12.5,500,0,0],z0,Tool \wobj:=Wobj_Part_0;
		MoveL Tr_meulage_motif_1_P125,[12.5,500,0,0],z0,Tool \wobj:=Wobj_Part_0;
		MoveL Tr_meulage_motif_1_P126,[12.5,500,0,0],z0,Tool \wobj:=Wobj_Part_0;
		MoveL Tr_meulage_motif_1_P127,[12.5,500,0,0],z0,Tool \wobj:=Wobj_Part_0;
		MoveL Tr_meulage_motif_1_P128,[12.5,500,0,0],z0,Tool \wobj:=Wobj_Part_0;
		MoveL Tr_meulage_motif_1_P129,[12.5,500,0,0],z0,Tool \wobj:=Wobj_Part_0;
		MoveL Tr_meulage_motif_1_P130,[12.5,500,0,0],z0,Tool \wobj:=Wobj_Part_0;
		MoveL Tr_meulage_motif_1_P131,[12.5,500,0,0],z0,Tool \wobj:=Wobj_Part_0;
		MoveL Tr_meulage_motif_1_P132,[12.5,500,0,0],z0,Tool \wobj:=Wobj_Part_0;
		MoveL Tr_meulage_motif_1_P133,[12.5,500,0,0],z0,Tool \wobj:=Wobj_Part_0;
		MoveL Tr_meulage_motif_1_P134,[12.5,500,0,0],z0,Tool \wobj:=Wobj_Part_0;
		MoveL Tr_meulage_motif_1_P135,[12.5,500,0,0],z0,Tool \wobj:=Wobj_Part_0;
		MoveL Tr_meulage_motif_1_P136,[12.5,500,0,0],z0,Tool \wobj:=Wobj_Part_0;
		MoveL Tr_meulage_motif_1_P137,[12.5,500,0,0],z0,Tool \wobj:=Wobj_Part_0;
		MoveL Tr_meulage_motif_1_P138,[12.5,500,0,0],z0,Tool \wobj:=Wobj_Part_0;
		MoveL Tr_meulage_motif_1_P139,[12.5,500,0,0],z0,Tool \wobj:=Wobj_Part_0;
		MoveL Tr_meulage_motif_1_P140,[12.5,500,0,0],z0,Tool \wobj:=Wobj_Part_0;
		MoveL Tr_meulage_motif_1_P141,[12.5,500,0,0],z0,Tool \wobj:=Wobj_Part_0;
		MoveL Tr_meulage_motif_1_P142,[12.5,500,0,0],z0,Tool \wobj:=Wobj_Part_0;
		MoveL Tr_meulage_motif_1_P143,[12.5,500,0,0],z0,Tool \wobj:=Wobj_Part_0;
		MoveL Tr_meulage_motif_1_P144,[12.5,500,0,0],z0,Tool \wobj:=Wobj_Part_0;
		MoveL Tr_meulage_motif_1_P145,[12.5,500,0,0],z0,Tool \wobj:=Wobj_Part_0;
		MoveL Tr_meulage_motif_1_P146,[12.5,500,0,0],z0,Tool \wobj:=Wobj_Part_0;
		MoveL Tr_meulage_motif_1_P147,[12.5,500,0,0],z0,Tool \wobj:=Wobj_Part_0;
		MoveL Tr_meulage_motif_1_P148,[12.5,500,0,0],z0,Tool \wobj:=Wobj_Part_0;
		MoveL Tr_meulage_motif_1_P149,[12.5,500,0,0],z0,Tool \wobj:=Wobj_Part_0;
		MoveL Tr_meulage_motif_1_P150,[12.5,500,0,0],z0,Tool \wobj:=Wobj_Part_0;
		MoveL Tr_meulage_motif_1_P151,[12.5,500,0,0],z0,Tool \wobj:=Wobj_Part_0;
		MoveL Tr_meulage_motif_1_P152,[12.5,500,0,0],z0,Tool \wobj:=Wobj_Part_0;
		MoveL Tr_meulage_motif_1_P153,[12.5,500,0,0],z0,Tool \wobj:=Wobj_Part_0;
		MoveL Tr_meulage_motif_1_P154,[12.5,500,0,0],z0,Tool \wobj:=Wobj_Part_0;
		MoveL Tr_meulage_motif_1_P155,[12.5,500,0,0],z0,Tool \wobj:=Wobj_Part_0;
		MoveL Tr_meulage_motif_1_P156,[12.5,500,0,0],z0,Tool \wobj:=Wobj_Part_0;
		MoveL Tr_meulage_motif_1_P157,[12.5,500,0,0],z0,Tool \wobj:=Wobj_Part_0;
		MoveL Tr_meulage_motif_1_P158,[12.5,500,0,0],z0,Tool \wobj:=Wobj_Part_0;
		MoveL Tr_meulage_motif_1_P159,[12.5,500,0,0],z0,Tool \wobj:=Wobj_Part_0;
		MoveL Tr_meulage_motif_1_P160,[12.5,500,0,0],z0,Tool \wobj:=Wobj_Part_0;
		MoveL Tr_meulage_motif_1_P161,[12.5,500,0,0],z0,Tool \wobj:=Wobj_Part_0;
		MoveL Tr_meulage_motif_1_P162,[12.5,500,0,0],z0,Tool \wobj:=Wobj_Part_0;
		MoveL Tr_meulage_motif_1_P163,[12.5,500,0,0],z0,Tool \wobj:=Wobj_Part_0;
		MoveL Tr_meulage_motif_1_P164,[12.5,500,0,0],z0,Tool \wobj:=Wobj_Part_0;
		MoveL Tr_meulage_motif_1_P165,[12.5,500,0,0],z0,Tool \wobj:=Wobj_Part_0;
		MoveL Tr_meulage_motif_1_P166,[12.5,500,0,0],z0,Tool \wobj:=Wobj_Part_0;
		MoveL Tr_meulage_motif_1_P167,[12.5,500,0,0],z0,Tool \wobj:=Wobj_Part_0;
		MoveL Tr_meulage_motif_1_P168,[12.5,500,0,0],z0,Tool \wobj:=Wobj_Part_0;
		MoveL Tr_meulage_motif_1_P169,[12.5,500,0,0],z0,Tool \wobj:=Wobj_Part_0;
		MoveL Tr_meulage_motif_1_P170,[12.5,500,0,0],z0,Tool \wobj:=Wobj_Part_0;
		MoveL Tr_meulage_motif_1_P171,[12.5,500,0,0],z0,Tool \wobj:=Wobj_Part_0;
		MoveL Tr_meulage_motif_1_P172,[12.5,500,0,0],z0,Tool \wobj:=Wobj_Part_0;
		MoveL Tr_meulage_motif_1_P173,[12.5,500,0,0],z0,Tool \wobj:=Wobj_Part_0;
		MoveL Tr_meulage_motif_1_P174,[12.5,500,0,0],z0,Tool \wobj:=Wobj_Part_0;
		MoveL Tr_meulage_motif_1_P175,[12.5,500,0,0],z0,Tool \wobj:=Wobj_Part_0;
		MoveL Tr_meulage_motif_1_P176,[12.5,500,0,0],z0,Tool \wobj:=Wobj_Part_0;
		MoveL Tr_meulage_motif_1_P177,[12.5,500,0,0],z0,Tool \wobj:=Wobj_Part_0;
		MoveL Tr_meulage_motif_1_P178,[12.5,500,0,0],z0,Tool \wobj:=Wobj_Part_0;
		MoveL Tr_meulage_motif_1_P179,[12.5,500,0,0],z0,Tool \wobj:=Wobj_Part_0;
		MoveL Tr_meulage_motif_1_P180,[12.5,500,0,0],z0,Tool \wobj:=Wobj_Part_0;
		MoveL Tr_meulage_motif_1_P181,[12.5,500,0,0],z0,Tool \wobj:=Wobj_Part_0;
		MoveL Tr_meulage_motif_1_P182,[12.5,500,0,0],z0,Tool \wobj:=Wobj_Part_0;
		MoveL Tr_meulage_motif_1_P183,[12.5,500,0,0],z0,Tool \wobj:=Wobj_Part_0;
		MoveL Tr_meulage_motif_1_P184,[12.5,500,0,0],z0,Tool \wobj:=Wobj_Part_0;
		MoveL Tr_meulage_motif_1_P185,[12.5,500,0,0],z0,Tool \wobj:=Wobj_Part_0;
		MoveL Tr_meulage_motif_1_P186,[12.5,500,0,0],z0,Tool \wobj:=Wobj_Part_0;
		MoveL Tr_meulage_motif_1_P187,[12.5,500,0,0],z0,Tool \wobj:=Wobj_Part_0;
		MoveL Tr_meulage_motif_1_P188,[12.5,500,0,0],z0,Tool \wobj:=Wobj_Part_0;
		MoveL Tr_meulage_motif_1_P189,[12.5,500,0,0],z0,Tool \wobj:=Wobj_Part_0;
		MoveL Tr_meulage_motif_1_P190,[12.5,500,0,0],z0,Tool \wobj:=Wobj_Part_0;
		MoveL Tr_meulage_motif_1_P191,[12.5,500,0,0],z0,Tool \wobj:=Wobj_Part_0;
		MoveL Tr_meulage_motif_1_P192,[12.5,500,0,0],z0,Tool \wobj:=Wobj_Part_0;
		MoveL Tr_meulage_motif_1_P193,[12.5,500,0,0],z0,Tool \wobj:=Wobj_Part_0;
		MoveL Tr_meulage_motif_1_P194,[12.5,500,0,0],z0,Tool \wobj:=Wobj_Part_0;
		MoveL Tr_meulage_motif_1_P195,[12.5,500,0,0],z0,Tool \wobj:=Wobj_Part_0;
		MoveL Tr_meulage_motif_1_P196,[12.5,500,0,0],z0,Tool \wobj:=Wobj_Part_0;
		MoveL Tr_meulage_motif_1_P197,[12.5,500,0,0],z0,Tool \wobj:=Wobj_Part_0;
		MoveL Tr_meulage_motif_1_P198,[12.5,500,0,0],z0,Tool \wobj:=Wobj_Part_0;
		MoveL Tr_meulage_motif_1_P199,[12.5,500,0,0],z0,Tool \wobj:=Wobj_Part_0;
		MoveL Tr_meulage_motif_1_P200,[12.5,500,0,0],z0,Tool \wobj:=Wobj_Part_0;
		MoveL Tr_meulage_motif_1_P201,[12.5,500,0,0],z0,Tool \wobj:=Wobj_Part_0;
		MoveL Tr_meulage_motif_1_P202,[12.5,500,0,0],z0,Tool \wobj:=Wobj_Part_0;
		MoveL Tr_meulage_motif_1_P203,[12.5,500,0,0],z0,Tool \wobj:=Wobj_Part_0;
		MoveL Tr_meulage_motif_1_P204,[12.5,500,0,0],z0,Tool \wobj:=Wobj_Part_0;
		MoveL Tr_meulage_motif_1_P205,[12.5,500,0,0],z0,Tool \wobj:=Wobj_Part_0;
		MoveL Tr_meulage_motif_1_P206,[12.5,500,0,0],z0,Tool \wobj:=Wobj_Part_0;
		MoveL Tr_meulage_motif_1_P207,[12.5,500,0,0],z0,Tool \wobj:=Wobj_Part_0;
		MoveL Tr_meulage_motif_1_P208,[12.5,500,0,0],z0,Tool \wobj:=Wobj_Part_0;
		MoveL Tr_meulage_motif_1_P209,[12.5,500,0,0],z0,Tool \wobj:=Wobj_Part_0;
		MoveL Tr_meulage_motif_1_P210,[12.5,500,0,0],z0,Tool \wobj:=Wobj_Part_0;
		MoveL Tr_meulage_motif_1_P211,[12.5,500,0,0],z0,Tool \wobj:=Wobj_Part_0;
		MoveL Tr_meulage_motif_1_P212,[12.5,500,0,0],z0,Tool \wobj:=Wobj_Part_0;
		MoveL Tr_meulage_motif_1_P213,[12.5,500,0,0],z0,Tool \wobj:=Wobj_Part_0;
		MoveL Tr_meulage_motif_1_P214,[12.5,500,0,0],z0,Tool \wobj:=Wobj_Part_0;
		MoveL Tr_meulage_motif_1_P215,[12.5,500,0,0],z0,Tool \wobj:=Wobj_Part_0;
		MoveL Tr_meulage_motif_1_P216,[12.5,500,0,0],z0,Tool \wobj:=Wobj_Part_0;
		MoveL Tr_meulage_motif_1_P217,[12.5,500,0,0],z0,Tool \wobj:=Wobj_Part_0;
		MoveL Tr_meulage_motif_1_P218,[12.5,500,0,0],z0,Tool \wobj:=Wobj_Part_0;
		MoveL Tr_meulage_motif_1_P219,[12.5,500,0,0],z0,Tool \wobj:=Wobj_Part_0;
		MoveL Tr_meulage_motif_1_P220,[12.5,500,0,0],z0,Tool \wobj:=Wobj_Part_0;
		MoveL Tr_meulage_motif_1_P221,[12.5,500,0,0],z0,Tool \wobj:=Wobj_Part_0;
		MoveL Tr_meulage_motif_1_P222,[12.5,500,0,0],z0,Tool \wobj:=Wobj_Part_0;
		MoveL Tr_meulage_motif_1_P223,[12.5,500,0,0],z0,Tool \wobj:=Wobj_Part_0;
		MoveL Tr_meulage_motif_1_P224,[12.5,500,0,0],z0,Tool \wobj:=Wobj_Part_0;
		MoveL Tr_meulage_motif_1_P225,[12.5,500,0,0],z0,Tool \wobj:=Wobj_Part_0;
		MoveL Tr_meulage_motif_1_P226,[12.5,500,0,0],z0,Tool \wobj:=Wobj_Part_0;
		MoveL Tr_meulage_motif_1_P227,[12.5,500,0,0],z0,Tool \wobj:=Wobj_Part_0;
		MoveL Tr_meulage_motif_1_P228,[12.5,500,0,0],z0,Tool \wobj:=Wobj_Part_0;
		MoveL Tr_meulage_motif_1_P229,[12.5,500,0,0],z0,Tool \wobj:=Wobj_Part_0;
		MoveL Tr_meulage_motif_1_P230,[12.5,500,0,0],z0,Tool \wobj:=Wobj_Part_0;
		MoveL Tr_meulage_motif_1_P231,[12.5,500,0,0],z0,Tool \wobj:=Wobj_Part_0;
		MoveL Tr_meulage_motif_1_P232,[12.5,500,0,0],z0,Tool \wobj:=Wobj_Part_0;
		MoveL Tr_meulage_motif_1_P233,[12.5,500,0,0],z0,Tool \wobj:=Wobj_Part_0;
		MoveL Tr_meulage_motif_1_P234,[12.5,500,0,0],z0,Tool \wobj:=Wobj_Part_0;
		MoveL Tr_meulage_motif_1_P235,[12.5,500,0,0],z0,Tool \wobj:=Wobj_Part_0;
		MoveL Tr_meulage_motif_1_P236,[12.5,500,0,0],z0,Tool \wobj:=Wobj_Part_0;
		MoveL Tr_meulage_motif_1_P237,[12.5,500,0,0],z0,Tool \wobj:=Wobj_Part_0;
		MoveL Tr_meulage_motif_1_P238,[12.5,500,0,0],z0,Tool \wobj:=Wobj_Part_0;
		MoveL Tr_meulage_motif_1_P239,[12.5,500,0,0],z0,Tool \wobj:=Wobj_Part_0;
		MoveL Tr_meulage_motif_1_P240,[12.5,500,0,0],z0,Tool \wobj:=Wobj_Part_0;
		MoveL Tr_meulage_motif_1_P241,[12.5,500,0,0],z0,Tool \wobj:=Wobj_Part_0;
		MoveL Tr_meulage_motif_1_P242,[12.5,500,0,0],z0,Tool \wobj:=Wobj_Part_0;
		MoveL Tr_meulage_motif_1_P243,[12.5,500,0,0],z0,Tool \wobj:=Wobj_Part_0;
		MoveL Tr_meulage_motif_1_P244,[12.5,500,0,0],z0,Tool \wobj:=Wobj_Part_0;
		MoveL Tr_meulage_motif_1_P245,[12.5,500,0,0],z0,Tool \wobj:=Wobj_Part_0;
		MoveL Tr_meulage_motif_1_P246,[12.5,500,0,0],z0,Tool \wobj:=Wobj_Part_0;
		MoveL Tr_meulage_motif_1_P247,[12.5,500,0,0],z0,Tool \wobj:=Wobj_Part_0;
		MoveL Tr_meulage_motif_1_P248,[12.5,500,0,0],z0,Tool \wobj:=Wobj_Part_0;
		MoveL Tr_meulage_motif_1_P249,[12.5,500,0,0],z0,Tool \wobj:=Wobj_Part_0;
		MoveL Tr_meulage_motif_1_P250,[12.5,500,0,0],z0,Tool \wobj:=Wobj_Part_0;
		MoveL Tr_meulage_motif_1_P251,[12.5,500,0,0],z0,Tool \wobj:=Wobj_Part_0;
		MoveL Tr_meulage_motif_1_P252,[12.5,500,0,0],z0,Tool \wobj:=Wobj_Part_0;
		MoveL Tr_meulage_motif_1_P253,[12.5,500,0,0],z0,Tool \wobj:=Wobj_Part_0;
		MoveL Tr_meulage_motif_1_P254,[12.5,500,0,0],z0,Tool \wobj:=Wobj_Part_0;
		MoveL Tr_meulage_motif_1_P255,[12.5,500,0,0],z0,Tool \wobj:=Wobj_Part_0;
		MoveL Tr_meulage_motif_1_P256,[12.5,500,0,0],z0,Tool \wobj:=Wobj_Part_0;
		MoveL Tr_meulage_motif_1_P257,[12.5,500,0,0],z0,Tool \wobj:=Wobj_Part_0;
		MoveL Tr_meulage_motif_1_P258,[12.5,500,0,0],z0,Tool \wobj:=Wobj_Part_0;
		MoveL Tr_meulage_motif_1_P259,[12.5,500,0,0],z0,Tool \wobj:=Wobj_Part_0;
		MoveL Tr_meulage_motif_1_P260,[12.5,500,0,0],z0,Tool \wobj:=Wobj_Part_0;
		MoveL Tr_meulage_motif_1_P261,[12.5,500,0,0],z0,Tool \wobj:=Wobj_Part_0;
		MoveL Tr_meulage_motif_1_P262,[12.5,500,0,0],z0,Tool \wobj:=Wobj_Part_0;
		MoveL Tr_meulage_motif_1_P263,[12.5,500,0,0],z0,Tool \wobj:=Wobj_Part_0;
		MoveL Tr_meulage_motif_1_P264,[12.5,500,0,0],z0,Tool \wobj:=Wobj_Part_0;
		MoveL Tr_meulage_motif_1_P265,[12.5,500,0,0],z0,Tool \wobj:=Wobj_Part_0;
		MoveL Tr_meulage_motif_1_P266,[12.5,500,0,0],z0,Tool \wobj:=Wobj_Part_0;
		MoveL Tr_meulage_motif_1_P267,[12.5,500,0,0],z0,Tool \wobj:=Wobj_Part_0;
		MoveL Tr_meulage_motif_1_P268,[12.5,500,0,0],z0,Tool \wobj:=Wobj_Part_0;
		MoveL Tr_meulage_motif_1_P269,[12.5,500,0,0],z0,Tool \wobj:=Wobj_Part_0;
		MoveL Tr_meulage_motif_1_P270,[12.5,500,0,0],z0,Tool \wobj:=Wobj_Part_0;
		MoveL Tr_meulage_motif_1_P271,[12.5,500,0,0],z0,Tool \wobj:=Wobj_Part_0;
		MoveL Tr_meulage_motif_1_P272,[12.5,500,0,0],z0,Tool \wobj:=Wobj_Part_0;
		MoveL Tr_meulage_motif_1_P273,[12.5,500,0,0],z0,Tool \wobj:=Wobj_Part_0;
		MoveL Tr_meulage_motif_1_P274,[12.5,500,0,0],z0,Tool \wobj:=Wobj_Part_0;
		MoveL Tr_meulage_motif_1_P275,[12.5,500,0,0],z0,Tool \wobj:=Wobj_Part_0;
		MoveL Tr_meulage_motif_1_P276,[12.5,500,0,0],z0,Tool \wobj:=Wobj_Part_0;
		MoveL Tr_meulage_motif_1_P277,[12.5,500,0,0],z0,Tool \wobj:=Wobj_Part_0;
		MoveL Tr_meulage_motif_1_P278,[12.5,500,0,0],z0,Tool \wobj:=Wobj_Part_0;
		MoveL Tr_meulage_motif_1_P279,[12.5,500,0,0],z0,Tool \wobj:=Wobj_Part_0;
		MoveL Tr_meulage_motif_1_P280,[12.5,500,0,0],z0,Tool \wobj:=Wobj_Part_0;
		MoveL Tr_meulage_motif_1_P281,[12.5,500,0,0],z0,Tool \wobj:=Wobj_Part_0;
		MoveL Tr_meulage_motif_1_P282,[12.5,500,0,0],z0,Tool \wobj:=Wobj_Part_0;
		MoveL Tr_meulage_motif_1_P283,[12.5,500,0,0],z0,Tool \wobj:=Wobj_Part_0;
		MoveL Tr_meulage_motif_1_P284,[12.5,500,0,0],z0,Tool \wobj:=Wobj_Part_0;
		MoveL Tr_meulage_motif_1_P285,[12.5,500,0,0],z0,Tool \wobj:=Wobj_Part_0;
		MoveL Tr_meulage_motif_1_P286,[12.5,500,0,0],z0,Tool \wobj:=Wobj_Part_0;
		MoveL Tr_meulage_motif_1_P287,[12.5,500,0,0],z0,Tool \wobj:=Wobj_Part_0;
		MoveL Tr_meulage_motif_1_P288,[12.5,500,0,0],z0,Tool \wobj:=Wobj_Part_0;
		MoveL Tr_meulage_motif_1_P289,[12.5,500,0,0],z0,Tool \wobj:=Wobj_Part_0;
		MoveL Tr_meulage_motif_1_P290,[12.5,500,0,0],z0,Tool \wobj:=Wobj_Part_0;
		MoveL Tr_meulage_motif_1_P291,[12.5,500,0,0],z0,Tool \wobj:=Wobj_Part_0;
		MoveL Tr_meulage_motif_1_P292,[12.5,500,0,0],z0,Tool \wobj:=Wobj_Part_0;
		MoveL Tr_meulage_motif_1_P293,[12.5,500,0,0],z0,Tool \wobj:=Wobj_Part_0;
		MoveL Tr_meulage_motif_1_P294,[12.5,500,0,0],z0,Tool \wobj:=Wobj_Part_0;
		MoveL Tr_meulage_motif_1_P295,[12.5,500,0,0],z0,Tool \wobj:=Wobj_Part_0;
		MoveL Tr_meulage_motif_1_P296,[12.5,500,0,0],z0,Tool \wobj:=Wobj_Part_0;
		MoveL Tr_meulage_motif_1_P297,[12.5,500,0,0],z0,Tool \wobj:=Wobj_Part_0;
		MoveL Tr_meulage_motif_1_P298,[12.5,500,0,0],z0,Tool \wobj:=Wobj_Part_0;
		MoveL Tr_meulage_motif_1_P299,[12.5,500,0,0],z0,Tool \wobj:=Wobj_Part_0;
		MoveL Tr_meulage_motif_1_P300,[12.5,500,0,0],z0,Tool \wobj:=Wobj_Part_0;
		MoveL Tr_meulage_motif_1_P301,[12.5,500,0,0],z0,Tool \wobj:=Wobj_Part_0;
		MoveL Tr_meulage_motif_1_P302,[12.5,500,0,0],z0,Tool \wobj:=Wobj_Part_0;
		MoveL Tr_meulage_motif_1_P303,[12.5,500,0,0],z0,Tool \wobj:=Wobj_Part_0;
		MoveL Tr_meulage_motif_1_P304,[12.5,500,0,0],z0,Tool \wobj:=Wobj_Part_0;
		MoveL Tr_meulage_motif_1_P305,[12.5,500,0,0],z0,Tool \wobj:=Wobj_Part_0;
		MoveL Tr_meulage_motif_1_P306,[12.5,500,0,0],z0,Tool \wobj:=Wobj_Part_0;
		MoveL Tr_meulage_motif_1_P307,[12.5,500,0,0],z0,Tool \wobj:=Wobj_Part_0;
		MoveL Tr_meulage_motif_1_P308,[12.5,500,0,0],z0,Tool \wobj:=Wobj_Part_0;
		MoveL Tr_meulage_motif_1_P309,[12.5,500,0,0],z0,Tool \wobj:=Wobj_Part_0;
		MoveL Tr_meulage_motif_1_P310,[12.5,500,0,0],z0,Tool \wobj:=Wobj_Part_0;
		MoveL Tr_meulage_motif_1_P311,[12.5,500,0,0],z0,Tool \wobj:=Wobj_Part_0;
		MoveL Tr_meulage_motif_1_P312,[12.5,500,0,0],z0,Tool \wobj:=Wobj_Part_0;
		MoveL Tr_meulage_motif_1_P313,[12.5,500,0,0],z0,Tool \wobj:=Wobj_Part_0;
		MoveL Tr_meulage_motif_1_P314,[12.5,500,0,0],z0,Tool \wobj:=Wobj_Part_0;
		MoveL Tr_meulage_motif_1_P315,[12.5,500,0,0],z0,Tool \wobj:=Wobj_Part_0;
		MoveL Tr_meulage_motif_1_P316,[12.5,500,0,0],z0,Tool \wobj:=Wobj_Part_0;
		MoveL Tr_meulage_motif_1_P317,[12.5,500,0,0],z0,Tool \wobj:=Wobj_Part_0;
		MoveL Tr_meulage_motif_1_P318,[12.5,500,0,0],z0,Tool \wobj:=Wobj_Part_0;
		MoveL Tr_meulage_motif_1_P319,[12.5,500,0,0],z0,Tool \wobj:=Wobj_Part_0;
		MoveL Tr_meulage_motif_1_P320,[12.5,500,0,0],z0,Tool \wobj:=Wobj_Part_0;
		MoveL Tr_meulage_motif_1_P321,[12.5,500,0,0],z0,Tool \wobj:=Wobj_Part_0;
		MoveL Tr_meulage_motif_1_P322,[12.5,500,0,0],z0,Tool \wobj:=Wobj_Part_0;
		MoveL Tr_meulage_motif_1_P323,[12.5,500,0,0],z0,Tool \wobj:=Wobj_Part_0;
		MoveL Tr_meulage_motif_1_P324,[12.5,500,0,0],z0,Tool \wobj:=Wobj_Part_0;
		MoveL Tr_meulage_motif_1_P325,[12.5,500,0,0],z0,Tool \wobj:=Wobj_Part_0;
		MoveL Tr_meulage_motif_1_P326,[12.5,500,0,0],z0,Tool \wobj:=Wobj_Part_0;
		MoveL Tr_meulage_motif_1_P327,[12.5,500,0,0],z0,Tool \wobj:=Wobj_Part_0;
		MoveL Tr_meulage_motif_1_P328,[12.5,500,0,0],z0,Tool \wobj:=Wobj_Part_0;
		MoveL Tr_meulage_motif_1_P329,[12.5,500,0,0],z0,Tool \wobj:=Wobj_Part_0;
		MoveL Tr_meulage_motif_1_P330,[12.5,500,0,0],z0,Tool \wobj:=Wobj_Part_0;
		MoveL Tr_meulage_motif_1_P331,[12.5,500,0,0],z0,Tool \wobj:=Wobj_Part_0;
		MoveL Tr_meulage_motif_1_P332,[12.5,500,0,0],z0,Tool \wobj:=Wobj_Part_0;
		MoveL Tr_meulage_motif_1_P333,[12.5,500,0,0],z0,Tool \wobj:=Wobj_Part_0;
		MoveL Tr_meulage_motif_1_P334,[12.5,500,0,0],z0,Tool \wobj:=Wobj_Part_0;
		MoveL Tr_meulage_motif_1_P335,[12.5,500,0,0],z0,Tool \wobj:=Wobj_Part_0;
		MoveJ Tr_meulage_motif_1_degg1,V500,Z0,Tool,\Wobj:=Wobj_Part_0;
		MoveJ Tr_meulage_motif_1_degg2,V2000,Z100,Tool,\Wobj:=Wobj_Part_0;
	ENDPROC
